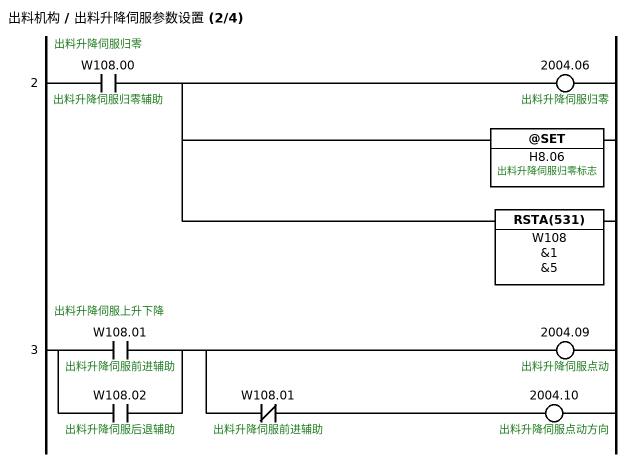
; [picture p360: 出料机构 / 出料升降伺服参数设置, rungs 2-3]
; rung 2: 出料升降伺服归零
LD W108.00  ; 出料升降伺服归零辅助
OUT 2004.06  ; 出料升降伺服归零
@SET H8.06  ; 出料升降伺服归零标志
RSTA(531) W108 &1 &5
; rung 3: 出料升降伺服上升下降
LD W108.01  ; 出料升降伺服前进辅助
OR W108.02  ; 出料升降伺服后退辅助
OUT 2004.09  ; 出料升降伺服点动
ANDNOT W108.01  ; 出料升降伺服前进辅助
OUT 2004.10  ; 出料升降伺服点动方向

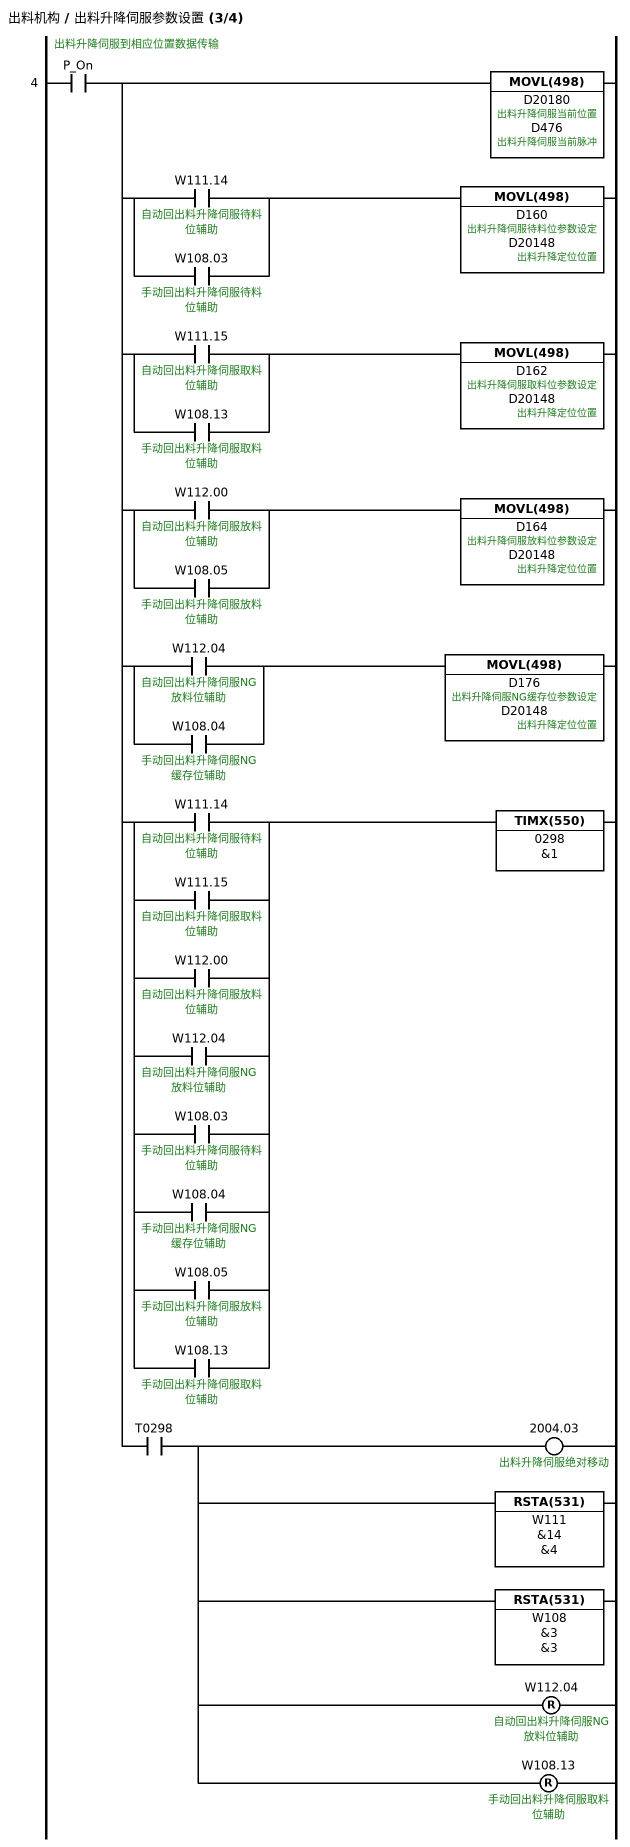
; rung 4: 出料升降伺服到相应位置数据传输
LD P_On
OUT TR0
MOVL(498) D20180 D476  ; 出料升降伺服当前位置, 出料升降伺服当前脉冲
LD W111.14  ; 自动回出料升降伺服待料位辅助
OR W108.03  ; 手动回出料升降伺服待料位辅助
ANDLD
MOVL(498) D160 D20148  ; 出料升降伺服待料位参数设定, 出料升降定位位置
LD TR0
LD W111.15  ; 自动回出料升降伺服取料位辅助
OR W108.13  ; 手动回出料升降伺服取料位辅助
ANDLD
MOVL(498) D162 D20148  ; 出料升降伺服取料位参数设定, 出料升降定位位置
LD TR0
LD W112.00  ; 自动回出料升降伺服放料位辅助
OR W108.05  ; 手动回出料升降伺服放料位辅助
ANDLD
MOVL(498) D164 D20148  ; 出料升降伺服放料位参数设定, 出料升降定位位置
LD TR0
LD W112.04  ; 自动回出料升降伺服NG放料位辅助
OR W108.04  ; 手动回出料升降伺服NG缓存位辅助
ANDLD
MOVL(498) D176 D20148  ; 出料升降伺服NG缓存位参数设定, 出料升降定位位置
LD TR0
LD W111.14  ; 自动回出料升降伺服待料位辅助
OR W111.15  ; 自动回出料升降伺服取料位辅助
OR W112.00  ; 自动回出料升降伺服放料位辅助
OR W112.04  ; 自动回出料升降伺服NG放料位辅助
OR W108.03  ; 手动回出料升降伺服待料位辅助
OR W108.04  ; 手动回出料升降伺服NG缓存位辅助
OR W108.05  ; 手动回出料升降伺服放料位辅助
OR W108.13  ; 手动回出料升降伺服取料位辅助
ANDLD
TIMX(550) 0298 &1
LD TR0
AND T0298
OUT 2004.03  ; 出料升降伺服绝对移动
RSTA(531) W111 &14 &4
RSTA(531) W108 &3 &3
RSET W112.04  ; 自动回出料升降伺服NG放料位辅助
RSET W108.13  ; 手动回出料升降伺服取料位辅助

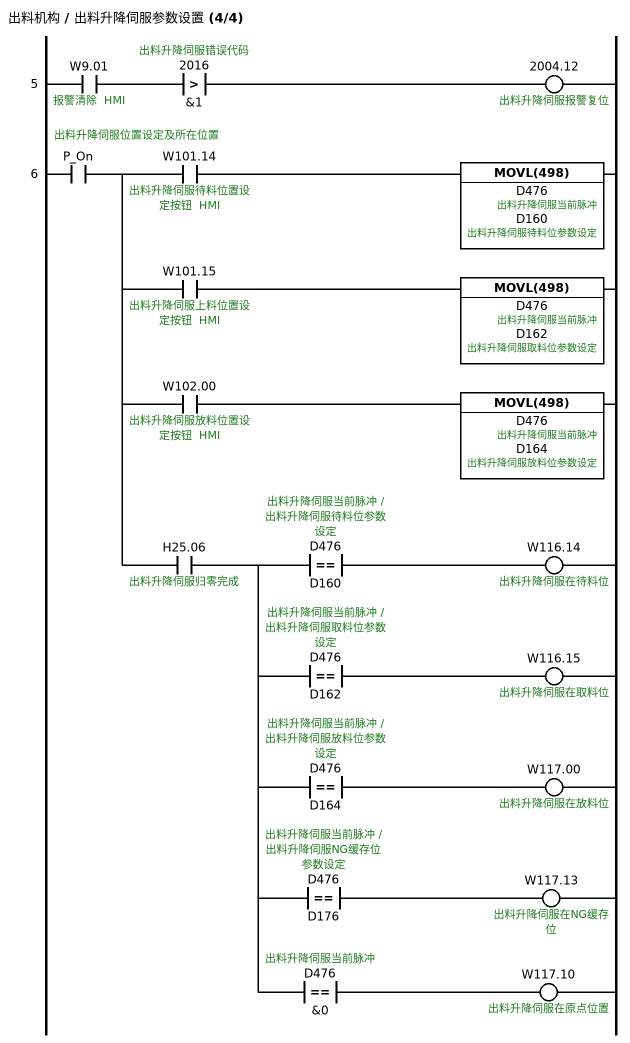
; rung 5
LD W9.01  ; 报警清除  HMI
AND>(320) 2016 &1  ; 出料升降伺服错误代码
OUT 2004.12  ; 出料升降伺服报警复位
; rung 6: 出料升降伺服位置设定及所在位置
LD P_On
OUT TR0
AND W101.14  ; 出料升降伺服待料位置设定按钮  HMI
MOVL(498) D476 D160  ; 出料升降伺服当前脉冲, 出料升降伺服待料位参数设定
LD TR0
AND W101.15  ; 出料升降伺服上料位置设定按钮  HMI
MOVL(498) D476 D162  ; 出料升降伺服当前脉冲, 出料升降伺服取料位参数设定
LD TR0
AND W102.00  ; 出料升降伺服放料位置设定按钮  HMI
MOVL(498) D476 D164  ; 出料升降伺服当前脉冲, 出料升降伺服放料位参数设定
LD TR0
AND H25.06  ; 出料升降伺服归零完成
OUT TR0
AND=SL(303) D476 D160  ; 出料升降伺服当前脉冲, 出料升降伺服待料位参数设定
OUT W116.14  ; 出料升降伺服在待料位
LD TR0
AND=SL(303) D476 D162  ; 出料升降伺服当前脉冲, 出料升降伺服取料位参数设定
OUT W116.15  ; 出料升降伺服在取料位
LD TR0
AND=SL(303) D476 D164  ; 出料升降伺服当前脉冲, 出料升降伺服放料位参数设定
OUT W117.00  ; 出料升降伺服在放料位
LD TR0
AND=SL(303) D476 D176  ; 出料升降伺服当前脉冲, 出料升降伺服NG缓存位参数设定
OUT W117.13  ; 出料升降伺服在NG缓存位
LD TR0
AND=SL(303) D476 &0  ; 出料升降伺服当前脉冲
OUT W117.10  ; 出料升降伺服在原点位置

### Section 出料旋转伺服参数设置

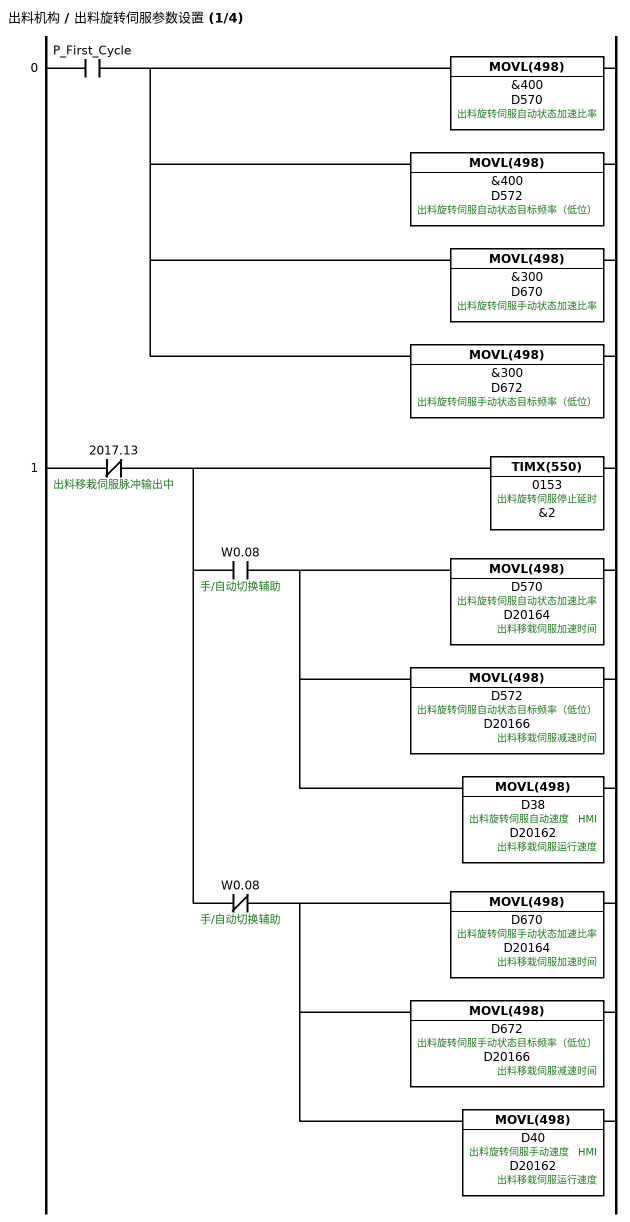
; rung 0
LD P_First_Cycle
MOVL(498) &400 D570  ; 出料旋转伺服自动状态加速比率
MOVL(498) &400 D572  ; 出料旋转伺服自动状态目标频率（低位）
MOVL(498) &300 D670  ; 出料旋转伺服手动状态加速比率
MOVL(498) &300 D672  ; 出料旋转伺服手动状态目标频率（低位）
; rung 1
LDNOT 2017.13  ; 出料移栽伺服脉冲输出中
OUT TR0
TIMX(550) 0153 &2  ; 出料旋转伺服停止延时
AND W0.08  ; 手/自动切换辅助
MOVL(498) D570 D20164  ; 出料旋转伺服自动状态加速比率, 出料移栽伺服加速时间
MOVL(498) D572 D20166  ; 出料旋转伺服自动状态目标频率（低位）, 出料移栽伺服减速时间
MOVL(498) D38 D20162  ; 出料旋转伺服自动速度   HMI, 出料移栽伺服运行速度
LD TR0
ANDNOT W0.08  ; 手/自动切换辅助
MOVL(498) D670 D20164  ; 出料旋转伺服手动状态加速比率, 出料移栽伺服加速时间
MOVL(498) D672 D20166  ; 出料旋转伺服手动状态目标频率（低位）, 出料移栽伺服减速时间
MOVL(498) D40 D20162  ; 出料旋转伺服手动速度   HMI, 出料移栽伺服运行速度

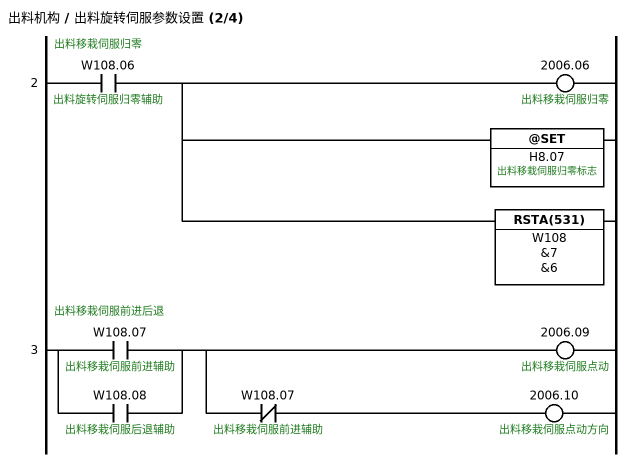
; rung 2: 出料移栽伺服归零
LD W108.06  ; 出料旋转伺服归零辅助
OUT 2006.06  ; 出料移栽伺服归零
@SET H8.07  ; 出料移栽伺服归零标志
RSTA(531) W108 &7 &6
; rung 3: 出料移栽伺服前进后退
LD W108.07  ; 出料移栽伺服前进辅助
OR W108.08  ; 出料移栽伺服后退辅助
OUT 2006.09  ; 出料移栽伺服点动
ANDNOT W108.07  ; 出料移栽伺服前进辅助
OUT 2006.10  ; 出料移栽伺服点动方向

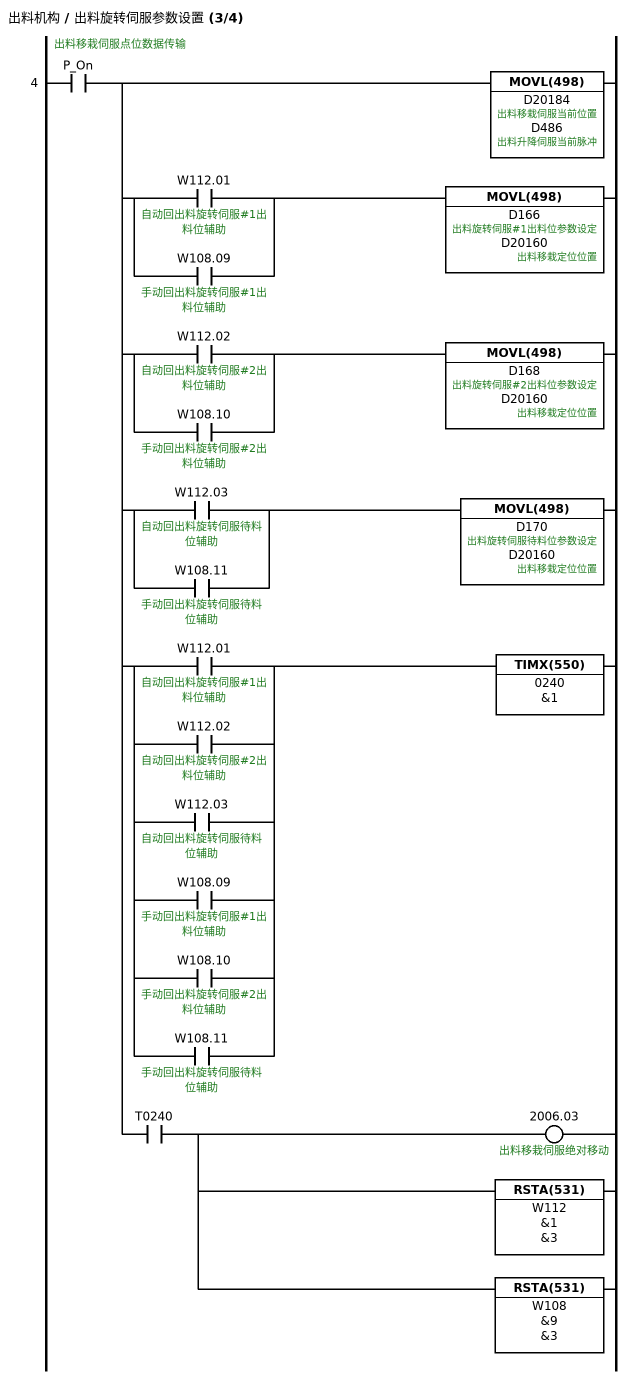
; rung 4: 出料移栽伺服点位数据传输
LD P_On
OUT TR0
MOVL(498) D20184 D486  ; 出料移栽伺服当前位置, 出料升降伺服当前脉冲
LD W112.01  ; 自动回出料旋转伺服#1出料位辅助
OR W108.09  ; 手动回出料旋转伺服#1出料位辅助
ANDLD
MOVL(498) D166 D20160  ; 出料旋转伺服#1出料位参数设定, 出料移栽定位位置
LD TR0
LD W112.02  ; 自动回出料旋转伺服#2出料位辅助
OR W108.10  ; 手动回出料旋转伺服#2出料位辅助
ANDLD
MOVL(498) D168 D20160  ; 出料旋转伺服#2出料位参数设定, 出料移栽定位位置
LD TR0
LD W112.03  ; 自动回出料旋转伺服待料位辅助
OR W108.11  ; 手动回出料旋转伺服待料位辅助
ANDLD
MOVL(498) D170 D20160  ; 出料旋转伺服待料位参数设定, 出料移栽定位位置
LD TR0
LD W112.01  ; 自动回出料旋转伺服#1出料位辅助
OR W112.02  ; 自动回出料旋转伺服#2出料位辅助
OR W112.03  ; 自动回出料旋转伺服待料位辅助
OR W108.09  ; 手动回出料旋转伺服#1出料位辅助
OR W108.10  ; 手动回出料旋转伺服#2出料位辅助
OR W108.11  ; 手动回出料旋转伺服待料位辅助
ANDLD
TIMX(550) 0240 &1
LD TR0
AND T0240
OUT 2006.03  ; 出料移栽伺服绝对移动
RSTA(531) W112 &1 &3
RSTA(531) W108 &9 &3

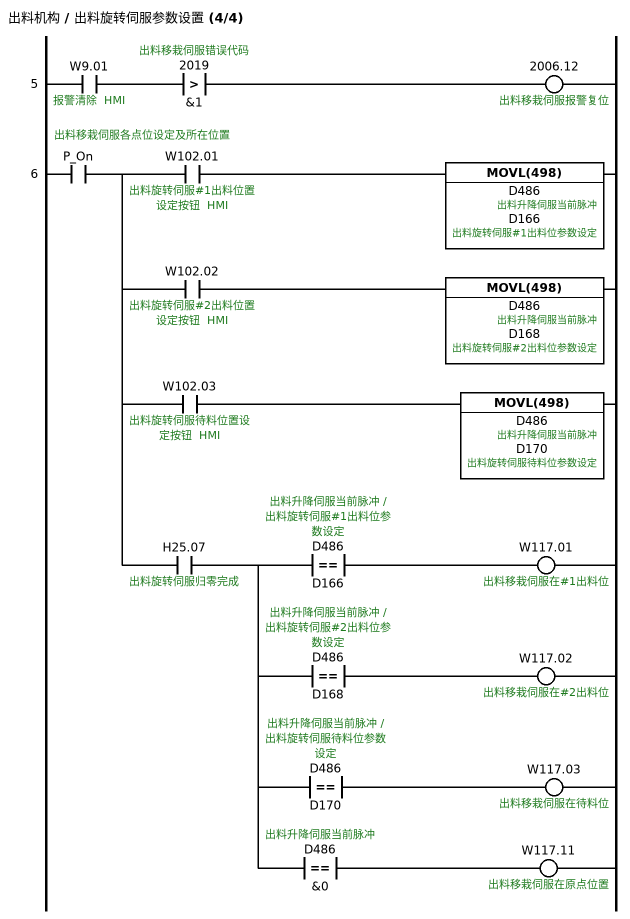
; rung 5
LD W9.01  ; 报警清除  HMI
AND>(320) 2019 &1  ; 出料移栽伺服错误代码
OUT 2006.12  ; 出料移栽伺服报警复位
; rung 6: 出料移栽伺服各点位设定及所在位置
LD P_On
OUT TR0
AND W102.01  ; 出料旋转伺服#1出料位置设定按钮  HMI
MOVL(498) D486 D166  ; 出料升降伺服当前脉冲, 出料旋转伺服#1出料位参数设定
LD TR0
AND W102.02  ; 出料旋转伺服#2出料位置设定按钮  HMI
MOVL(498) D486 D168  ; 出料升降伺服当前脉冲, 出料旋转伺服#2出料位参数设定
LD TR0
AND W102.03  ; 出料旋转伺服待料位置设定按钮  HMI
MOVL(498) D486 D170  ; 出料升降伺服当前脉冲, 出料旋转伺服待料位参数设定
LD TR0
AND H25.07  ; 出料旋转伺服归零完成
OUT TR0
AND=SL(303) D486 D166  ; 出料升降伺服当前脉冲, 出料旋转伺服#1出料位参数设定
OUT W117.01  ; 出料移栽伺服在#1出料位
LD TR0
AND=SL(303) D486 D168  ; 出料升降伺服当前脉冲, 出料旋转伺服#2出料位参数设定
OUT W117.02  ; 出料移栽伺服在#2出料位
LD TR0
AND=SL(303) D486 D170  ; 出料升降伺服当前脉冲, 出料旋转伺服待料位参数设定
OUT W117.03  ; 出料移栽伺服在待料位
LD TR0
AND=SL(303) D486 &0  ; 出料升降伺服当前脉冲
OUT W117.11  ; 出料移栽伺服在原点位置

### Section _4_框架信号对接

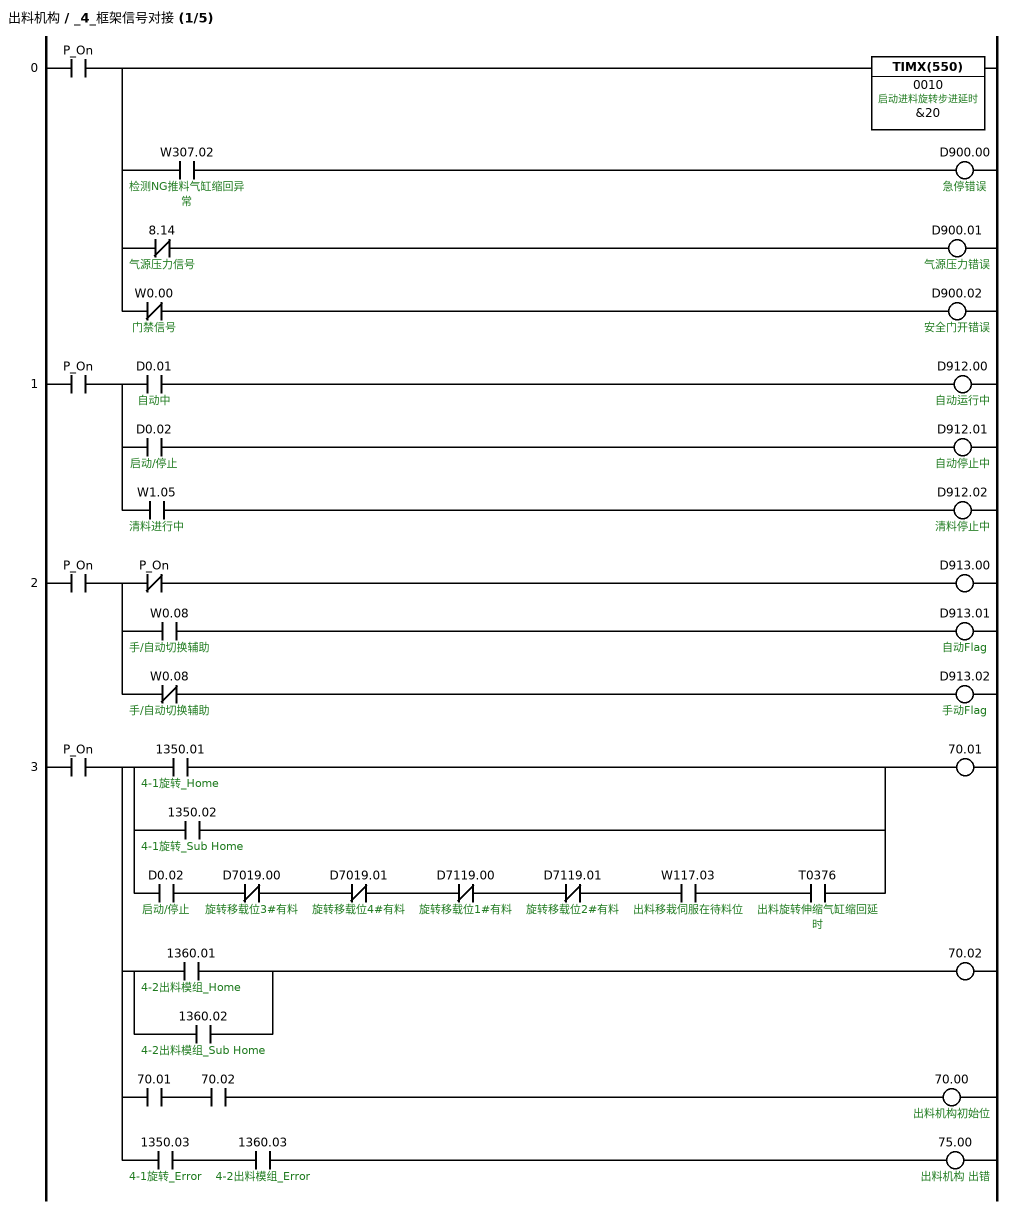
; rung 0
LD P_On
OUT TR0
TIMX(550) 0010 &20  ; 启动进料旋转步进延时
AND W307.02  ; 检测NG推料气缸缩回异常
OUT D900.00  ; 急停错误
LD TR0
ANDNOT 8.14  ; 气源压力信号
OUT D900.01  ; 气源压力错误
LD TR0
ANDNOT W0.00  ; 门禁信号
OUT D900.02  ; 安全门开错误
; rung 1
LD P_On
OUT TR0
AND D0.01  ; 自动中
OUT D912.00  ; 自动运行中
LD TR0
AND D0.02  ; 启动/停止
OUT D912.01  ; 自动停止中
LD TR0
AND W1.05  ; 清料进行中
OUT D912.02  ; 清料停止中
; rung 2
LD P_On
OUT TR0
ANDNOT P_On
OUT D913.00
LD TR0
AND W0.08  ; 手/自动切换辅助
OUT D913.01  ; 自动Flag
LD TR0
ANDNOT W0.08  ; 手/自动切换辅助
OUT D913.02  ; 手动Flag
; rung 3
LD P_On
OUT TR0
LD 1350.01  ; 4-1旋转_Home
OR 1350.02  ; 4-1旋转_Sub Home
LD D0.02  ; 启动/停止
ANDNOT D7019.00  ; 旋转移载位3#有料
ANDNOT D7019.01  ; 旋转移载位4#有料
ANDNOT D7119.00  ; 旋转移载位1#有料
ANDNOT D7119.01  ; 旋转移载位2#有料
AND W117.03  ; 出料移栽伺服在待料位
AND T0376  ; 出料旋转伸缩气缸缩回延时
ORLD
ANDLD
OUT 70.01
LD TR0
LD 1360.01  ; 4-2出料模组_Home
OR 1360.02  ; 4-2出料模组_Sub Home
ANDLD
OUT 70.02
LD TR0
AND 70.01
AND 70.02
OUT 70.00  ; 出料机构初始位
LD TR0
AND 1350.03  ; 4-1旋转_Error
AND 1360.03  ; 4-2出料模组_Error
OUT 75.00  ; 出料机构 出错

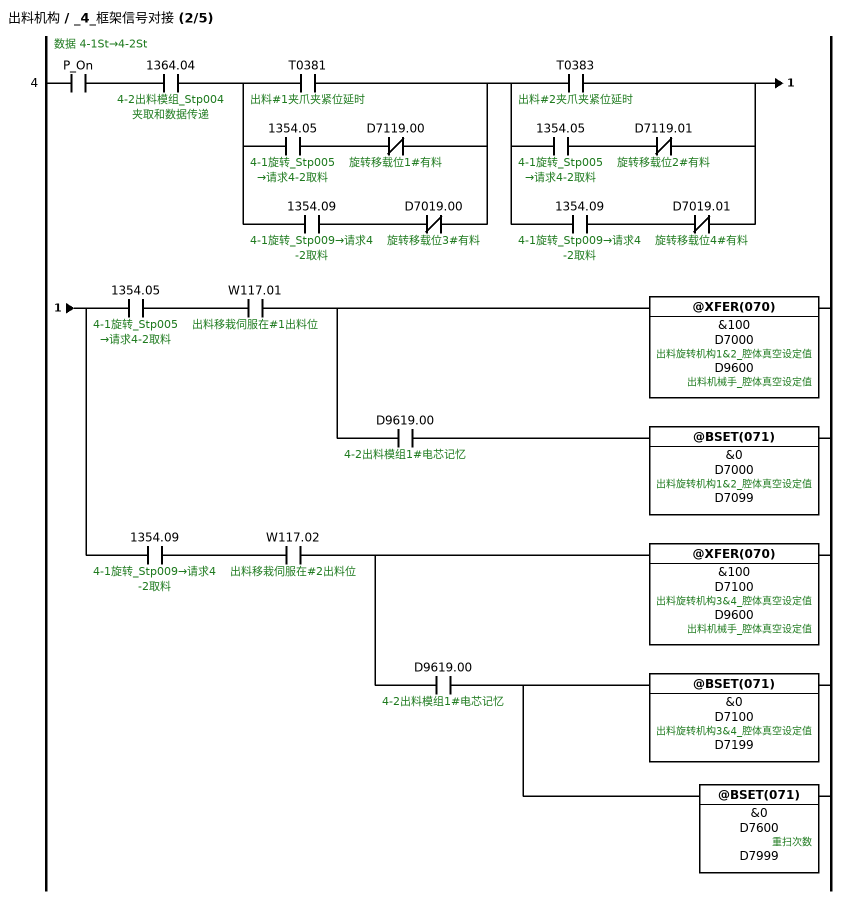
; rung 4: 数据 4-1St→4-2St
LD P_On
AND 1364.04  ; 4-2出料模组_Stp004 夹取和数据传递
LD T0381  ; 出料#1夹爪夹紧位延时
LD 1354.05  ; 4-1旋转_Stp005 →请求4-2取料
ANDNOT D7119.00  ; 旋转移载位1#有料
ORLD
LD 1354.09  ; 4-1旋转_Stp009→请求4-2取料
ANDNOT D7019.00  ; 旋转移载位3#有料
ORLD
ANDLD
LD T0383  ; 出料#2夹爪夹紧位延时
LD 1354.05  ; 4-1旋转_Stp005 →请求4-2取料
ANDNOT D7119.01  ; 旋转移载位2#有料
ORLD
LD 1354.09  ; 4-1旋转_Stp009→请求4-2取料
ANDNOT D7019.01  ; 旋转移载位4#有料
ORLD
ANDLD
OUT TR0
AND 1354.05  ; 4-1旋转_Stp005 →请求4-2取料
AND W117.01  ; 出料移栽伺服在#1出料位
@XFER(070) &100 D7000 D9600  ; 出料旋转机构1&2_腔体真空设定值, 出料机械手_腔体真空设定值
AND D9619.00  ; 4-2出料模组1#电芯记忆
@BSET(071) &0 D7000 D7099  ; 出料旋转机构1&2_腔体真空设定值
LD TR0
AND 1354.09  ; 4-1旋转_Stp009→请求4-2取料
AND W117.02  ; 出料移栽伺服在#2出料位
@XFER(070) &100 D7100 D9600  ; 出料旋转机构3&4_腔体真空设定值, 出料机械手_腔体真空设定值
AND D9619.00  ; 4-2出料模组1#电芯记忆
@BSET(071) &0 D7100 D7199  ; 出料旋转机构3&4_腔体真空设定值
@BSET(071) &0 D7600 D7999  ; 重扫次数

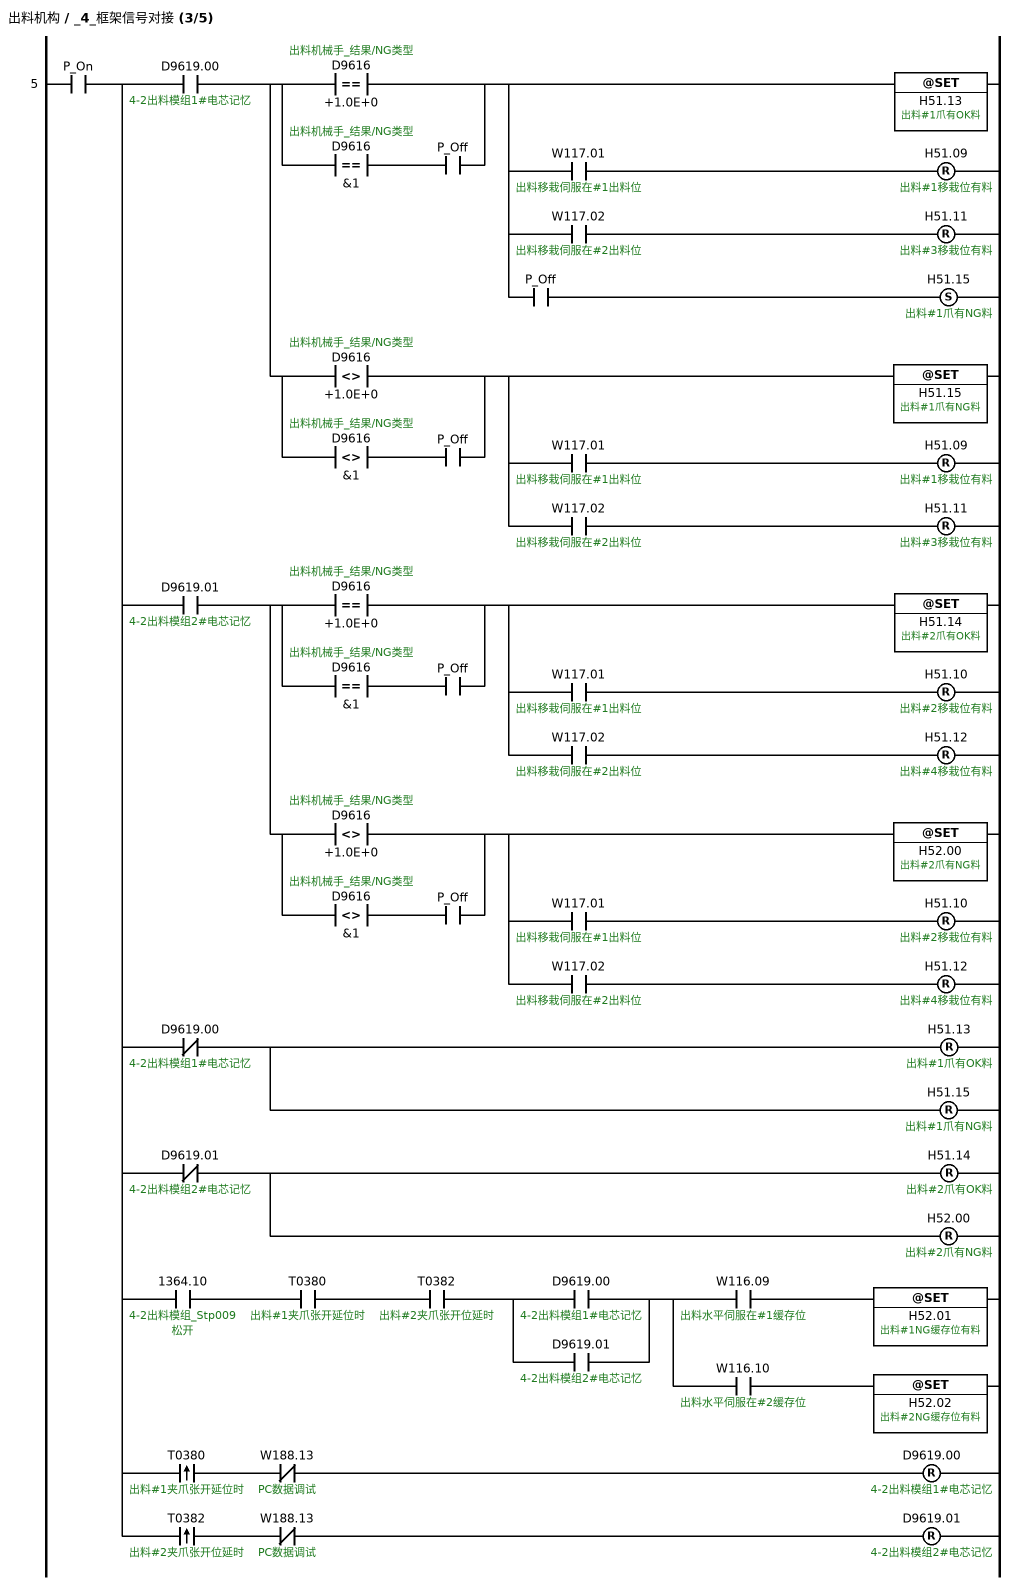
; rung 5
LD P_On
OUT TR0
AND D9619.00  ; 4-2出料模组1#电芯记忆
OUT TR1
LD=F(329) D9616 +1.0E+0  ; 出料机械手_结果/NG类型
LD=(300) D9616 &1  ; 出料机械手_结果/NG类型
AND P_Off
ORLD
ANDLD
OUT TR2
@SET H51.13  ; 出料#1爪有OK料
AND W117.01  ; 出料移栽伺服在#1出料位
RSET H51.09  ; 出料#1移栽位有料
LD TR2
AND W117.02  ; 出料移栽伺服在#2出料位
RSET H51.11  ; 出料#3移栽位有料
LD TR2
AND P_Off
SET H51.15  ; 出料#1爪有NG料
LD TR1
LD<>F(330) D9616 +1.0E+0  ; 出料机械手_结果/NG类型
LD<>(305) D9616 &1  ; 出料机械手_结果/NG类型
AND P_Off
ORLD
ANDLD
OUT TR1
@SET H51.15  ; 出料#1爪有NG料
AND W117.01  ; 出料移栽伺服在#1出料位
RSET H51.09  ; 出料#1移栽位有料
LD TR1
AND W117.02  ; 出料移栽伺服在#2出料位
RSET H51.11  ; 出料#3移栽位有料
LD TR0
AND D9619.01  ; 4-2出料模组2#电芯记忆
OUT TR1
LD=F(329) D9616 +1.0E+0  ; 出料机械手_结果/NG类型
LD=(300) D9616 &1  ; 出料机械手_结果/NG类型
AND P_Off
ORLD
ANDLD
OUT TR2
@SET H51.14  ; 出料#2爪有OK料
AND W117.01  ; 出料移栽伺服在#1出料位
RSET H51.10  ; 出料#2移栽位有料
LD TR2
AND W117.02  ; 出料移栽伺服在#2出料位
RSET H51.12  ; 出料#4移栽位有料
LD TR1
LD<>F(330) D9616 +1.0E+0  ; 出料机械手_结果/NG类型
LD<>(305) D9616 &1  ; 出料机械手_结果/NG类型
AND P_Off
ORLD
ANDLD
OUT TR1
@SET H52.00  ; 出料#2爪有NG料
AND W117.01  ; 出料移栽伺服在#1出料位
RSET H51.10  ; 出料#2移栽位有料
LD TR1
AND W117.02  ; 出料移栽伺服在#2出料位
RSET H51.12  ; 出料#4移栽位有料
LD TR0
ANDNOT D9619.00  ; 4-2出料模组1#电芯记忆
RSET H51.13  ; 出料#1爪有OK料
RSET H51.15  ; 出料#1爪有NG料
LD TR0
ANDNOT D9619.01  ; 4-2出料模组2#电芯记忆
RSET H51.14  ; 出料#2爪有OK料
RSET H52.00  ; 出料#2爪有NG料
LD TR0
AND 1364.10  ; 4-2出料模组_Stp009 松开
AND T0380  ; 出料#1夹爪张开延位时
AND T0382  ; 出料#2夹爪张开位延时
LD D9619.00  ; 4-2出料模组1#电芯记忆
OR D9619.01  ; 4-2出料模组2#电芯记忆
ANDLD
OUT TR1
AND W116.09  ; 出料水平伺服在#1缓存位
@SET H52.01  ; 出料#1NG缓存位有料
LD TR1
AND W116.10  ; 出料水平伺服在#2缓存位
@SET H52.02  ; 出料#2NG缓存位有料
LD TR0
@AND T0380  ; 出料#1夹爪张开延位时
ANDNOT W188.13  ; PC数据调试
RSET D9619.00  ; 4-2出料模组1#电芯记忆
LD TR0
@AND T0382  ; 出料#2夹爪张开位延时
ANDNOT W188.13  ; PC数据调试
RSET D9619.01  ; 4-2出料模组2#电芯记忆

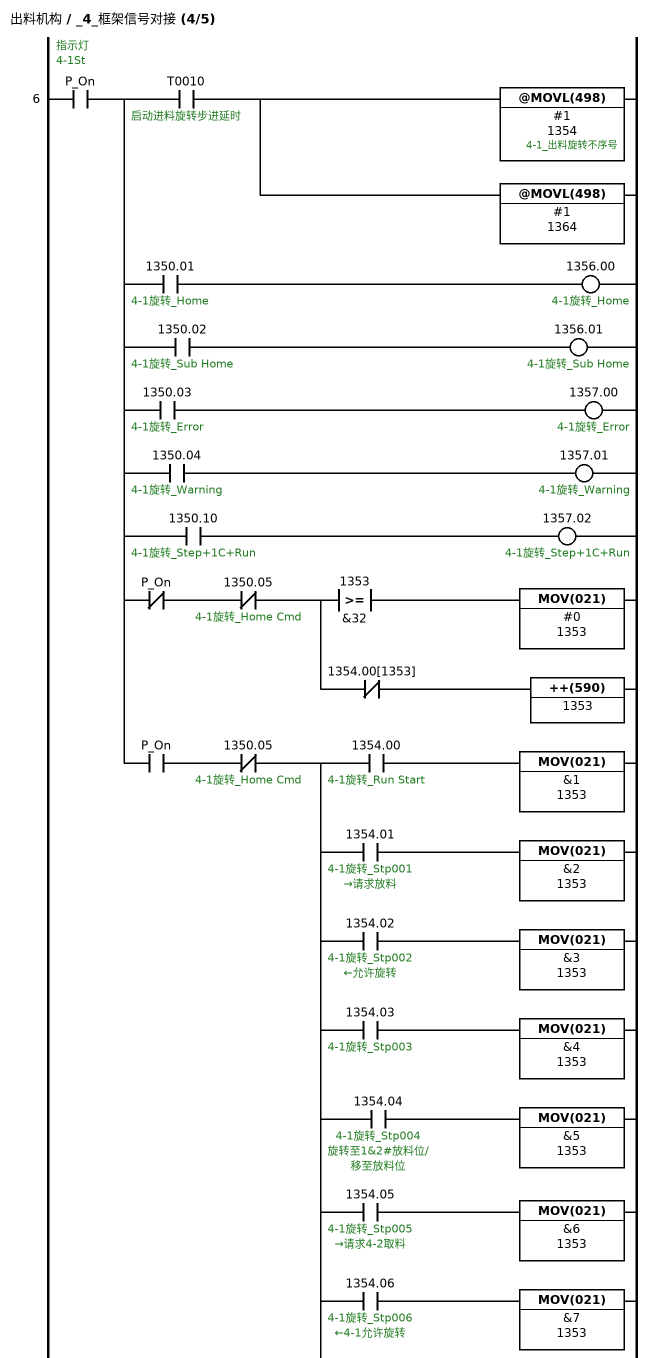

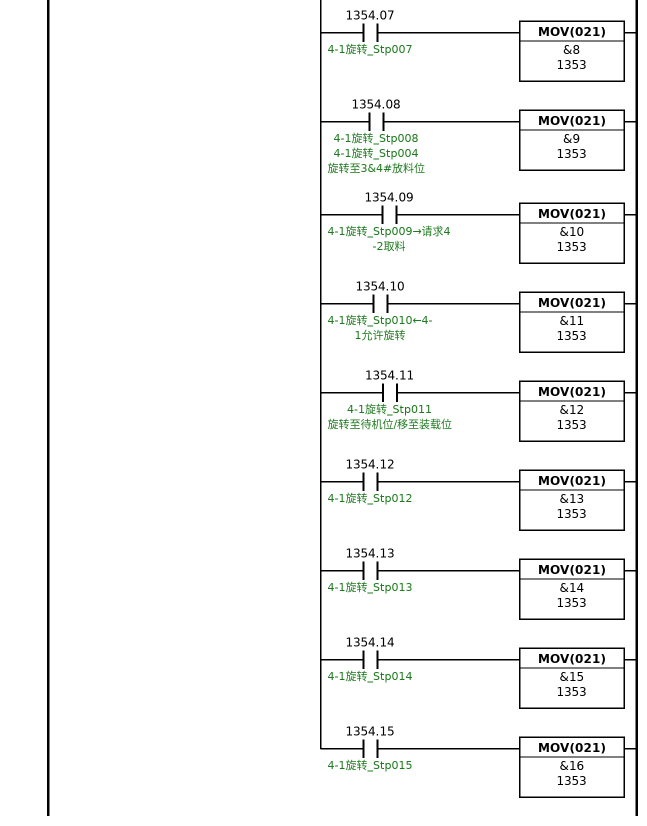
; rung 6: 指示灯 / 4-1St
LD P_On
OUT TR0
AND T0010  ; 启动进料旋转步进延时
@MOVL(498) #1 1354  ; 4-1_出料旋转不序号
@MOVL(498) #1 1364
LD TR0
AND 1350.01  ; 4-1旋转_Home
OUT 1356.00  ; 4-1旋转_Home
LD TR0
AND 1350.02  ; 4-1旋转_Sub Home
OUT 1356.01  ; 4-1旋转_Sub Home
LD TR0
AND 1350.03  ; 4-1旋转_Error
OUT 1357.00  ; 4-1旋转_Error
LD TR0
AND 1350.04  ; 4-1旋转_Warning
OUT 1357.01  ; 4-1旋转_Warning
LD TR0
AND 1350.10  ; 4-1旋转_Step+1C+Run
OUT 1357.02  ; 4-1旋转_Step+1C+Run
LD TR0
ANDNOT P_On
ANDNOT 1350.05  ; 4-1旋转_Home Cmd
OUT TR1
AND>=(325) 1353 &32
MOV(021) #0 1353
LD TR1
ANDNOT 1354.00[1353]
++(590) 1353
LD TR0
AND P_On
ANDNOT 1350.05  ; 4-1旋转_Home Cmd
OUT TR0
AND 1354.00  ; 4-1旋转_Run Start
MOV(021) &1 1353
LD TR0
AND 1354.01  ; 4-1旋转_Stp001 →请求放料
MOV(021) &2 1353
LD TR0
AND 1354.02  ; 4-1旋转_Stp002 ←允许旋转
MOV(021) &3 1353
LD TR0
AND 1354.03  ; 4-1旋转_Stp003
MOV(021) &4 1353
LD TR0
AND 1354.04  ; 4-1旋转_Stp004 旋转至1&2#放料位/移至放料位
MOV(021) &5 1353
LD TR0
AND 1354.05  ; 4-1旋转_Stp005 →请求4-2取料
MOV(021) &6 1353
LD TR0
AND 1354.06  ; 4-1旋转_Stp006 ←4-1允许旋转
MOV(021) &7 1353
LD TR0
AND 1354.07  ; 4-1旋转_Stp007
MOV(021) &8 1353
LD TR0
AND 1354.08  ; 4-1旋转_Stp008 4-1旋转_Stp004 旋转至3&4#放料位
MOV(021) &9 1353
LD TR0
AND 1354.09  ; 4-1旋转_Stp009→请求4-2取料
MOV(021) &10 1353
LD TR0
AND 1354.10  ; 4-1旋转_Stp010←4-1允许旋转
MOV(021) &11 1353
LD TR0
AND 1354.11  ; 4-1旋转_Stp011 旋转至待机位/移至装载位
MOV(021) &12 1353
LD TR0
AND 1354.12  ; 4-1旋转_Stp012
MOV(021) &13 1353
LD TR0
AND 1354.13  ; 4-1旋转_Stp013
MOV(021) &14 1353
LD TR0
AND 1354.14  ; 4-1旋转_Stp014
MOV(021) &15 1353
LD TR0
AND 1354.15  ; 4-1旋转_Stp015
MOV(021) &16 1353

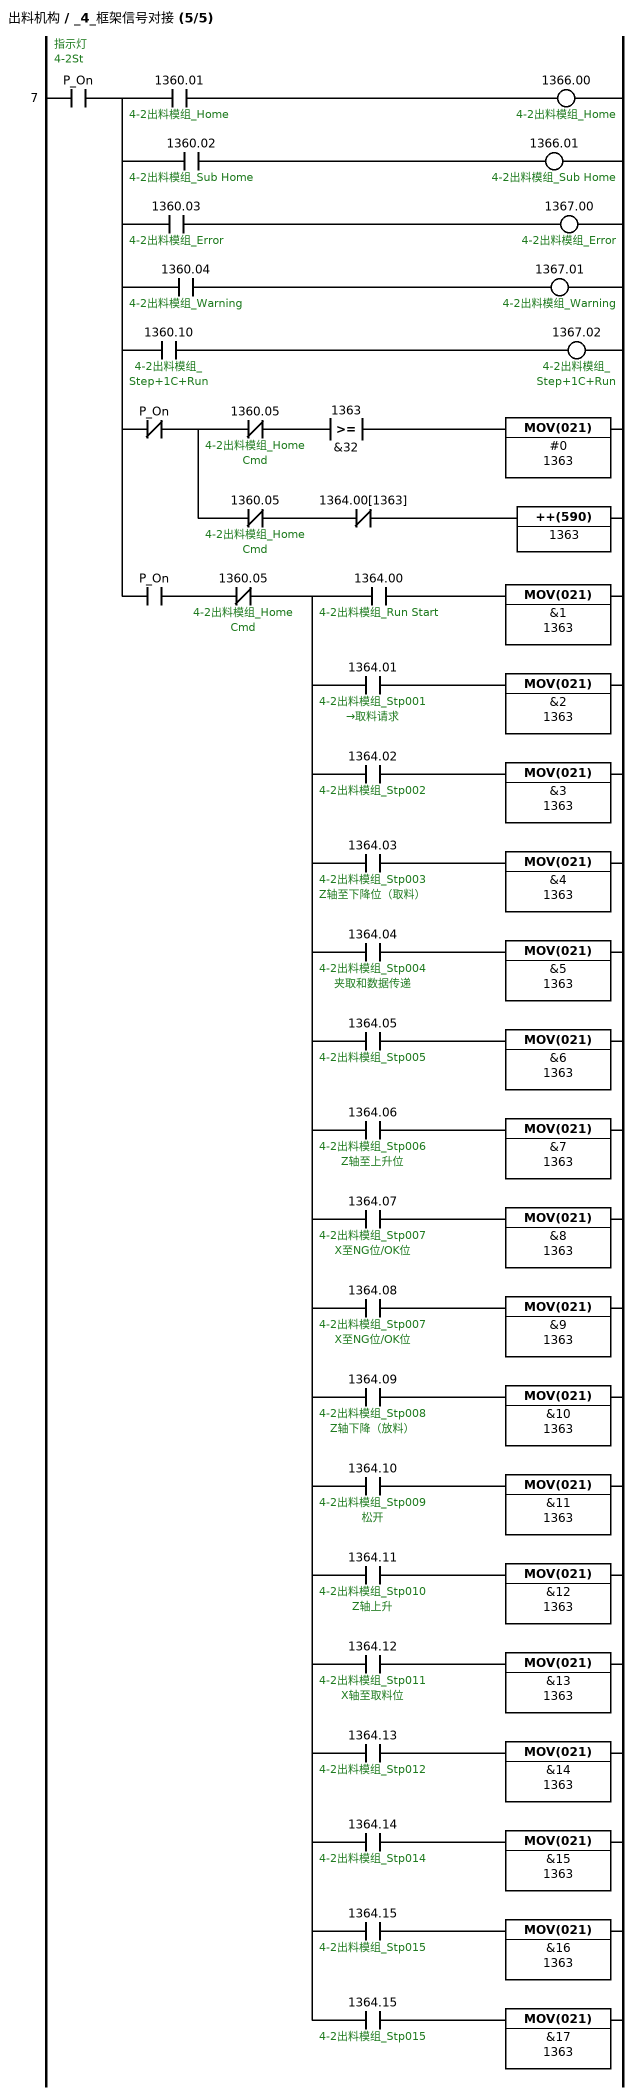
; rung 7: 指示灯 / 4-2St
LD P_On
OUT TR0
AND 1360.01  ; 4-2出料模组_Home
OUT 1366.00  ; 4-2出料模组_Home
LD TR0
AND 1360.02  ; 4-2出料模组_Sub Home
OUT 1366.01  ; 4-2出料模组_Sub Home
LD TR0
AND 1360.03  ; 4-2出料模组_Error
OUT 1367.00  ; 4-2出料模组_Error
LD TR0
AND 1360.04  ; 4-2出料模组_Warning
OUT 1367.01  ; 4-2出料模组_Warning
LD TR0
AND 1360.10  ; 4-2出料模组_Step+1C+Run
OUT 1367.02  ; 4-2出料模组_Step+1C+Run
LD TR0
ANDNOT P_On
OUT TR1
ANDNOT 1360.05  ; 4-2出料模组_Home Cmd
AND>=(325) 1363 &32
MOV(021) #0 1363
LD TR1
ANDNOT 1360.05  ; 4-2出料模组_Home Cmd
ANDNOT 1364.00[1363]
++(590) 1363
LD TR0
AND P_On
ANDNOT 1360.05  ; 4-2出料模组_Home Cmd
OUT TR0
AND 1364.00  ; 4-2出料模组_Run Start
MOV(021) &1 1363
LD TR0
AND 1364.01  ; 4-2出料模组_Stp001 →取料请求
MOV(021) &2 1363
LD TR0
AND 1364.02  ; 4-2出料模组_Stp002
MOV(021) &3 1363
LD TR0
AND 1364.03  ; 4-2出料模组_Stp003 Z轴至下降位（取料）
MOV(021) &4 1363
LD TR0
AND 1364.04  ; 4-2出料模组_Stp004 夹取和数据传递
MOV(021) &5 1363
LD TR0
AND 1364.05  ; 4-2出料模组_Stp005
MOV(021) &6 1363
LD TR0
AND 1364.06  ; 4-2出料模组_Stp006 Z轴至上升位
MOV(021) &7 1363
LD TR0
AND 1364.07  ; 4-2出料模组_Stp007 X至NG位/OK位
MOV(021) &8 1363
LD TR0
AND 1364.08  ; 4-2出料模组_Stp007 X至NG位/OK位
MOV(021) &9 1363
LD TR0
AND 1364.09  ; 4-2出料模组_Stp008 Z轴下降（放料）
MOV(021) &10 1363
LD TR0
AND 1364.10  ; 4-2出料模组_Stp009 松开
MOV(021) &11 1363
LD TR0
AND 1364.11  ; 4-2出料模组_Stp010 Z轴上升
MOV(021) &12 1363
LD TR0
AND 1364.12  ; 4-2出料模组_Stp011 X轴至取料位
MOV(021) &13 1363
LD TR0
AND 1364.13  ; 4-2出料模组_Stp012
MOV(021) &14 1363
LD TR0
AND 1364.14  ; 4-2出料模组_Stp014
MOV(021) &15 1363
LD TR0
AND 1364.15  ; 4-2出料模组_Stp015
MOV(021) &16 1363
LD TR0
AND 1364.15  ; 4-2出料模组_Stp015
MOV(021) &17 1363

### Section _4_1出料旋转自动

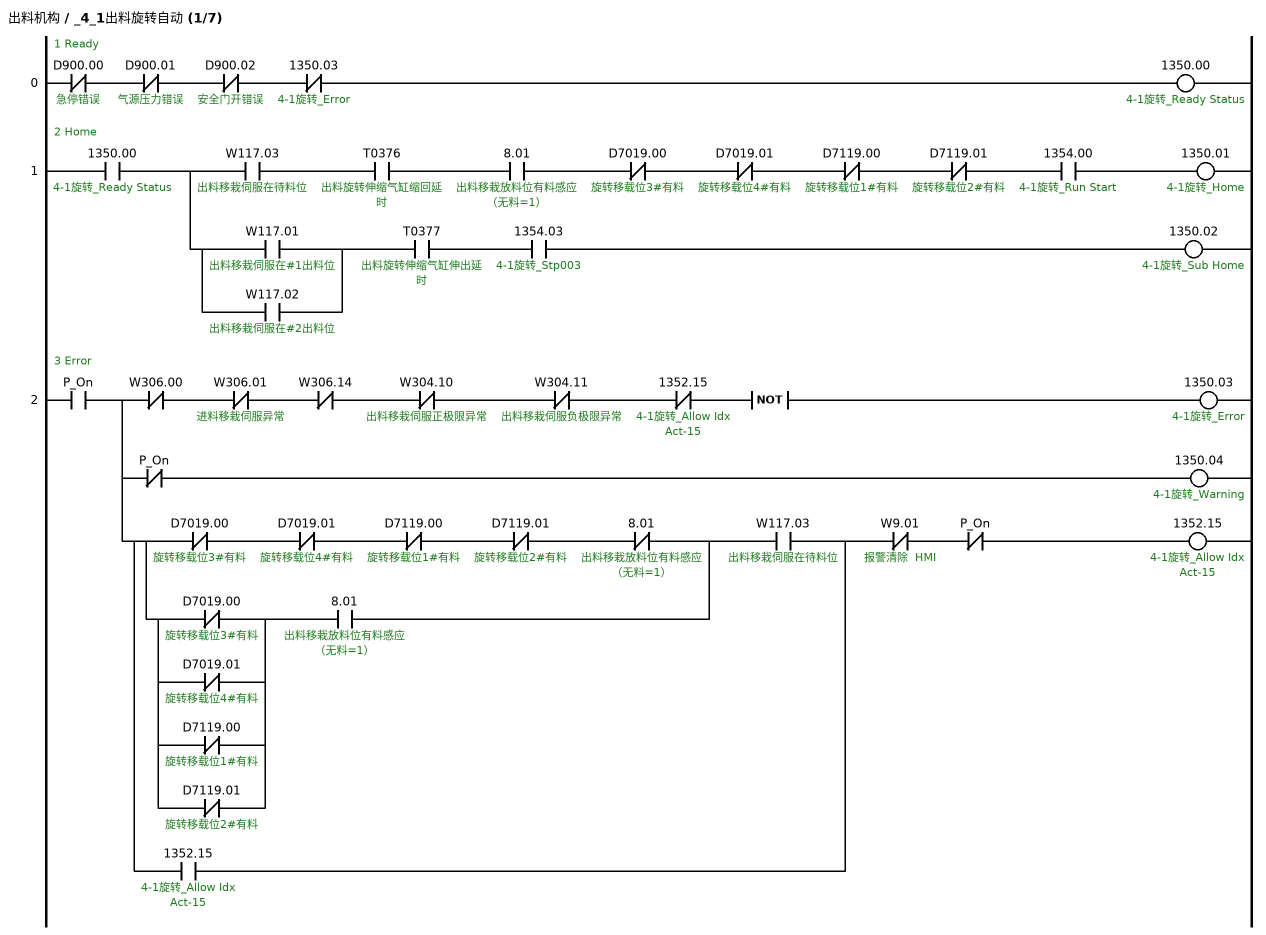
; rung 0: 1 Ready
LDNOT D900.00  ; 急停错误
ANDNOT D900.01  ; 气源压力错误
ANDNOT D900.02  ; 安全门开错误
ANDNOT 1350.03  ; 4-1旋转_Error
OUT 1350.00  ; 4-1旋转_Ready Status
; rung 1: 2 Home
LD 1350.00  ; 4-1旋转_Ready Status
OUT TR0
AND W117.03  ; 出料移栽伺服在待料位
AND T0376  ; 出料旋转伸缩气缸缩回延时
AND 8.01  ; 出料移栽放料位有料感应（无料=1）
ANDNOT D7019.00  ; 旋转移载位3#有料
ANDNOT D7019.01  ; 旋转移载位4#有料
ANDNOT D7119.00  ; 旋转移载位1#有料
ANDNOT D7119.01  ; 旋转移载位2#有料
AND 1354.00  ; 4-1旋转_Run Start
OUT 1350.01  ; 4-1旋转_Home
LD TR0
LD W117.01  ; 出料移栽伺服在#1出料位
OR W117.02  ; 出料移栽伺服在#2出料位
ANDLD
AND T0377  ; 出料旋转伸缩气缸伸出延时
AND 1354.03  ; 4-1旋转_Stp003
OUT 1350.02  ; 4-1旋转_Sub Home
; rung 2: 3 Error
LD P_On
OUT TR0
ANDNOT W306.00
ANDNOT W306.01  ; 进料移栽伺服异常
ANDNOT W306.14
ANDNOT W304.10  ; 出料移栽伺服正极限异常
ANDNOT W304.11  ; 出料移栽伺服负极限异常
ANDNOT 1352.15  ; 4-1旋转_Allow Idx Act-15
NOT(520)
OUT 1350.03  ; 4-1旋转_Error
LD TR0
ANDNOT P_On
OUT 1350.04  ; 4-1旋转_Warning
LD TR0
LDNOT D7019.00  ; 旋转移载位3#有料
ANDNOT D7019.01  ; 旋转移载位4#有料
ANDNOT D7119.00  ; 旋转移载位1#有料
ANDNOT D7119.01  ; 旋转移载位2#有料
ANDNOT 8.01  ; 出料移栽放料位有料感应（无料=1）
LDNOT D7019.00  ; 旋转移载位3#有料
ORNOT D7019.01  ; 旋转移载位4#有料
ORNOT D7119.00  ; 旋转移载位1#有料
ORNOT D7119.01  ; 旋转移载位2#有料
AND 8.01  ; 出料移栽放料位有料感应（无料=1）
ORLD
AND W117.03  ; 出料移栽伺服在待料位
OR 1352.15  ; 4-1旋转_Allow Idx Act-15
ANDLD
ANDNOT W9.01  ; 报警清除  HMI
ANDNOT P_On
OUT 1352.15  ; 4-1旋转_Allow Idx Act-15

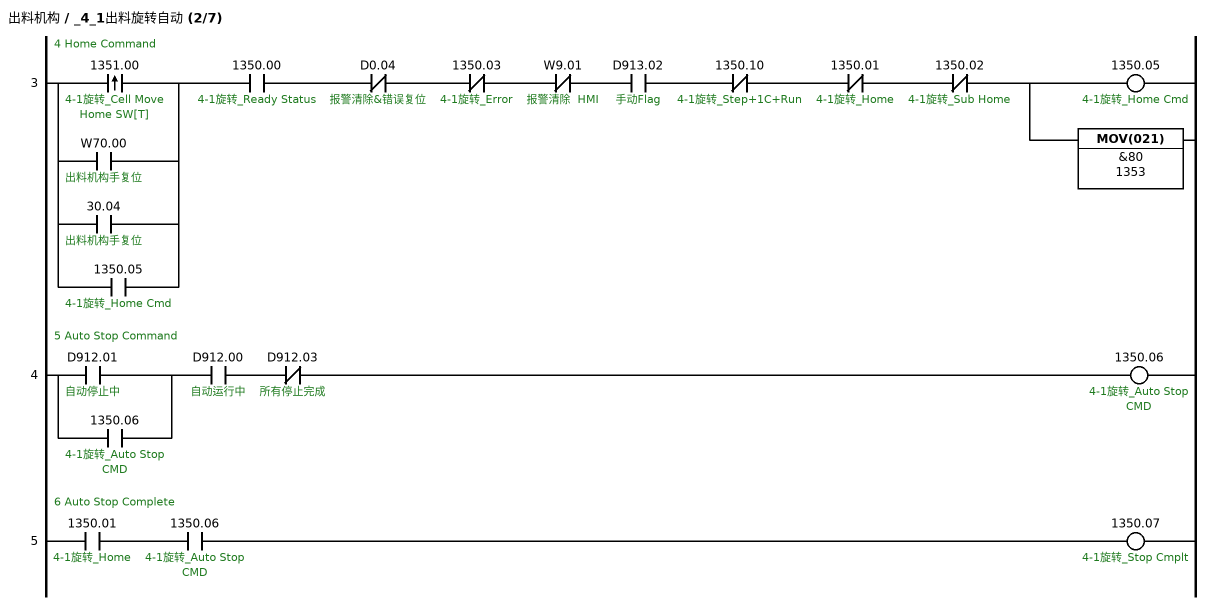
; rung 3: 4 Home Command
@LD 1351.00  ; 4-1旋转_Cell Move Home SW[T]
OR W70.00  ; 出料机构手复位
OR 30.04  ; 出料机构手复位
OR 1350.05  ; 4-1旋转_Home Cmd
AND 1350.00  ; 4-1旋转_Ready Status
ANDNOT D0.04  ; 报警清除&错误复位
ANDNOT 1350.03  ; 4-1旋转_Error
ANDNOT W9.01  ; 报警清除  HMI
AND D913.02  ; 手动Flag
ANDNOT 1350.10  ; 4-1旋转_Step+1C+Run
ANDNOT 1350.01  ; 4-1旋转_Home
ANDNOT 1350.02  ; 4-1旋转_Sub Home
OUT 1350.05  ; 4-1旋转_Home Cmd
MOV(021) &80 1353
; rung 4: 5 Auto Stop Command
LD D912.01  ; 自动停止中
OR 1350.06  ; 4-1旋转_Auto Stop CMD
AND D912.00  ; 自动运行中
ANDNOT D912.03  ; 所有停止完成
OUT 1350.06  ; 4-1旋转_Auto Stop CMD
; rung 5: 6 Auto Stop Complete
LD 1350.01  ; 4-1旋转_Home
AND 1350.06  ; 4-1旋转_Auto Stop CMD
OUT 1350.07  ; 4-1旋转_Stop Cmplt

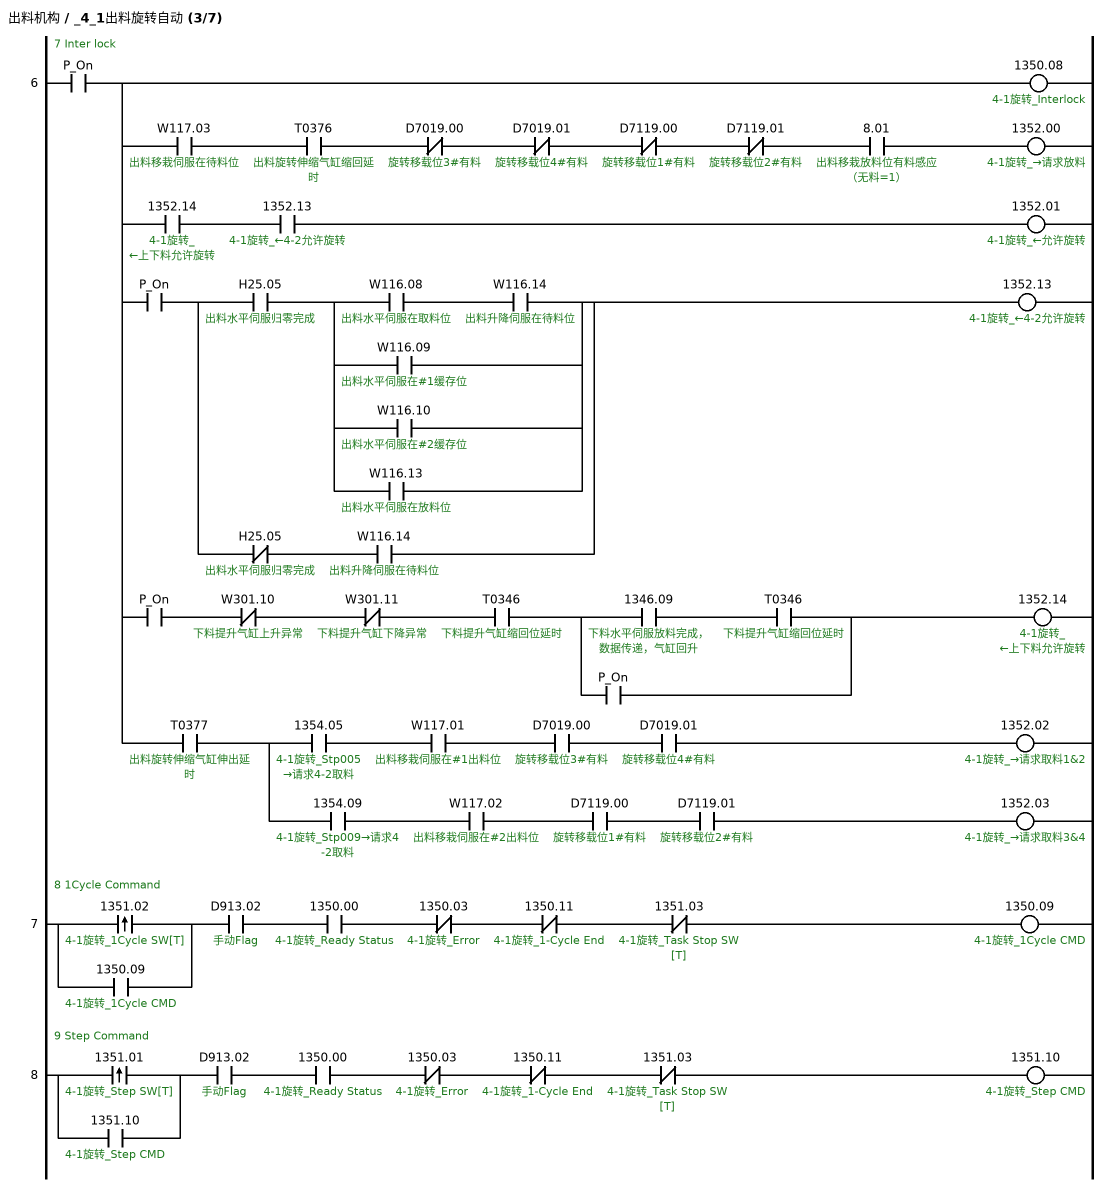
; rung 6: 7 Inter lock
LD P_On
OUT TR0
OUT 1350.08  ; 4-1旋转_Interlock
AND W117.03  ; 出料移栽伺服在待料位
AND T0376  ; 出料旋转伸缩气缸缩回延时
ANDNOT D7019.00  ; 旋转移载位3#有料
ANDNOT D7019.01  ; 旋转移载位4#有料
ANDNOT D7119.00  ; 旋转移载位1#有料
ANDNOT D7119.01  ; 旋转移载位2#有料
AND 8.01  ; 出料移栽放料位有料感应（无料=1）
OUT 1352.00  ; 4-1旋转_→请求放料
LD TR0
AND 1352.14  ; 4-1旋转_←上下料允许旋转
AND 1352.13  ; 4-1旋转_←4-2允许旋转
OUT 1352.01  ; 4-1旋转_←允许旋转
LD TR0
AND P_On
LD H25.05  ; 出料水平伺服归零完成
LD W116.08  ; 出料水平伺服在取料位
AND W116.14  ; 出料升降伺服在待料位
OR W116.09  ; 出料水平伺服在#1缓存位
OR W116.10  ; 出料水平伺服在#2缓存位
OR W116.13  ; 出料水平伺服在放料位
ANDLD
LDNOT H25.05  ; 出料水平伺服归零完成
AND W116.14  ; 出料升降伺服在待料位
ORLD
ANDLD
OUT 1352.13  ; 4-1旋转_←4-2允许旋转
LD TR0
AND P_On
ANDNOT W301.10  ; 下料提升气缸上升异常
ANDNOT W301.11  ; 下料提升气缸下降异常
AND T0346  ; 下料提升气缸缩回位延时
LD 1346.09  ; 下料水平伺服放料完成，数据传递，气缸回升
AND T0346  ; 下料提升气缸缩回位延时
OR P_On
ANDLD
OUT 1352.14  ; 4-1旋转_←上下料允许旋转
LD TR0
AND T0377  ; 出料旋转伸缩气缸伸出延时
OUT TR0
AND 1354.05  ; 4-1旋转_Stp005 →请求4-2取料
AND W117.01  ; 出料移栽伺服在#1出料位
AND D7019.00  ; 旋转移载位3#有料
AND D7019.01  ; 旋转移载位4#有料
OUT 1352.02  ; 4-1旋转_→请求取料1&2
LD TR0
AND 1354.09  ; 4-1旋转_Stp009→请求4-2取料
AND W117.02  ; 出料移栽伺服在#2出料位
AND D7119.00  ; 旋转移载位1#有料
AND D7119.01  ; 旋转移载位2#有料
OUT 1352.03  ; 4-1旋转_→请求取料3&4
; rung 7: 8 1Cycle Command
@LD 1351.02  ; 4-1旋转_1Cycle SW[T]
OR 1350.09  ; 4-1旋转_1Cycle CMD
AND D913.02  ; 手动Flag
AND 1350.00  ; 4-1旋转_Ready Status
ANDNOT 1350.03  ; 4-1旋转_Error
ANDNOT 1350.11  ; 4-1旋转_1-Cycle End
ANDNOT 1351.03  ; 4-1旋转_Task Stop SW [T]
OUT 1350.09  ; 4-1旋转_1Cycle CMD
; rung 8: 9 Step Command
@LD 1351.01  ; 4-1旋转_Step SW[T]
OR 1351.10  ; 4-1旋转_Step CMD
AND D913.02  ; 手动Flag
AND 1350.00  ; 4-1旋转_Ready Status
ANDNOT 1350.03  ; 4-1旋转_Error
ANDNOT 1350.11  ; 4-1旋转_1-Cycle End
ANDNOT 1351.03  ; 4-1旋转_Task Stop SW [T]
OUT 1351.10  ; 4-1旋转_Step CMD

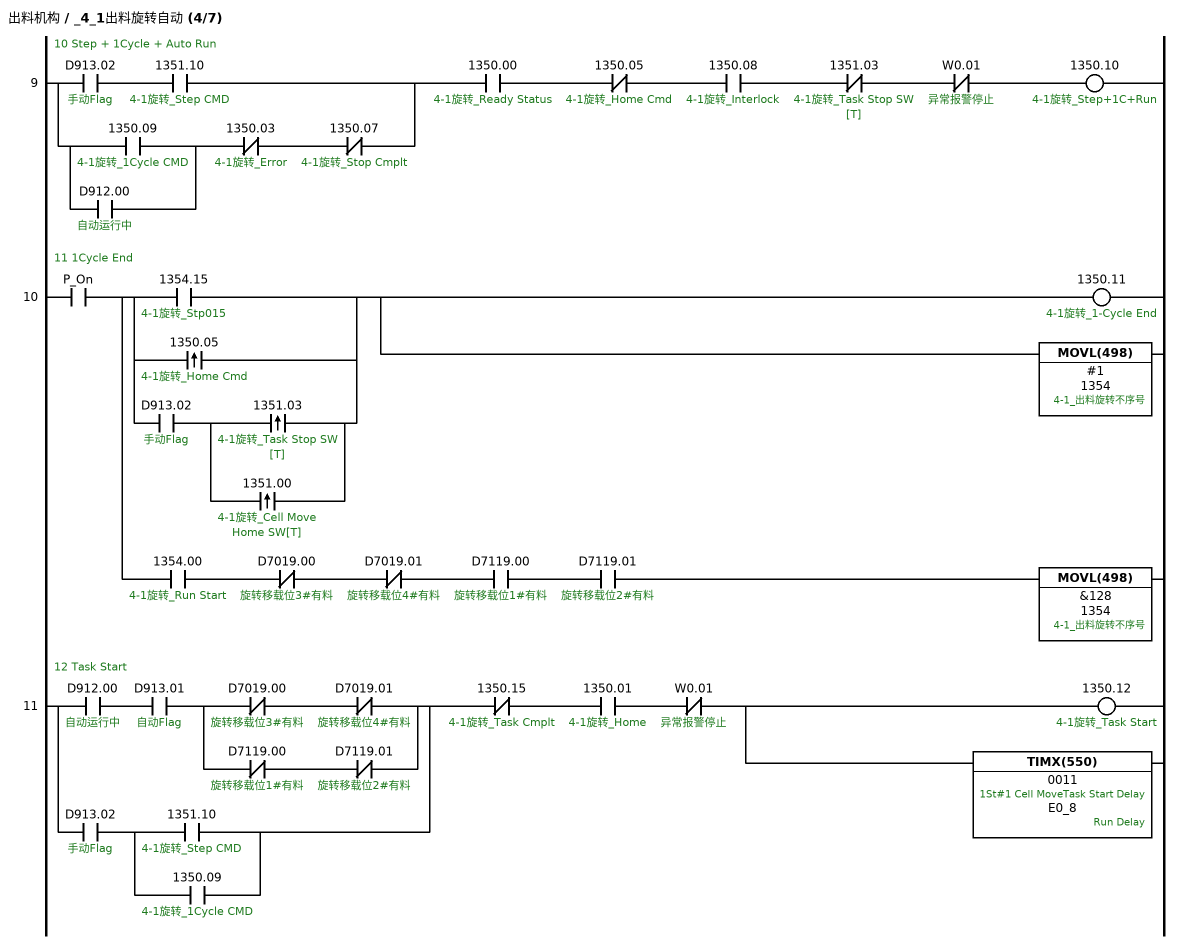
; rung 9: 10 Step + 1Cycle + Auto Run
LD D913.02  ; 手动Flag
AND 1351.10  ; 4-1旋转_Step CMD
LD 1350.09  ; 4-1旋转_1Cycle CMD
OR D912.00  ; 自动运行中
ANDNOT 1350.03  ; 4-1旋转_Error
ANDNOT 1350.07  ; 4-1旋转_Stop Cmplt
ORLD
AND 1350.00  ; 4-1旋转_Ready Status
ANDNOT 1350.05  ; 4-1旋转_Home Cmd
AND 1350.08  ; 4-1旋转_Interlock
ANDNOT 1351.03  ; 4-1旋转_Task Stop SW [T]
ANDNOT W0.01  ; 异常报警停止
OUT 1350.10  ; 4-1旋转_Step+1C+Run
; rung 10: 11 1Cycle End
LD P_On
OUT TR0
LD 1354.15  ; 4-1旋转_Stp015
@OR 1350.05  ; 4-1旋转_Home Cmd
LD D913.02  ; 手动Flag
@LD 1351.03  ; 4-1旋转_Task Stop SW [T]
@OR 1351.00  ; 4-1旋转_Cell Move Home SW[T]
ANDLD
ORLD
ANDLD
OUT 1350.11  ; 4-1旋转_1-Cycle End
MOVL(498) #1 1354  ; 4-1_出料旋转不序号
LD TR0
AND 1354.00  ; 4-1旋转_Run Start
ANDNOT D7019.00  ; 旋转移载位3#有料
ANDNOT D7019.01  ; 旋转移载位4#有料
AND D7119.00  ; 旋转移载位1#有料
AND D7119.01  ; 旋转移载位2#有料
MOVL(498) &128 1354  ; 4-1_出料旋转不序号
; rung 11: 12 Task Start
LD D912.00  ; 自动运行中
AND D913.01  ; 自动Flag
LDNOT D7019.00  ; 旋转移载位3#有料
ANDNOT D7019.01  ; 旋转移载位4#有料
LDNOT D7119.00  ; 旋转移载位1#有料
ANDNOT D7119.01  ; 旋转移载位2#有料
ORLD
ANDLD
LD D913.02  ; 手动Flag
LD 1351.10  ; 4-1旋转_Step CMD
OR 1350.09  ; 4-1旋转_1Cycle CMD
ANDLD
ORLD
ANDNOT 1350.15  ; 4-1旋转_Task Cmplt
AND 1350.01  ; 4-1旋转_Home
ANDNOT W0.01  ; 异常报警停止
OUT 1350.12  ; 4-1旋转_Task Start
TIMX(550) 0011 E0_8  ; Run Delay, 1St#1 Cell MoveTask Start Delay

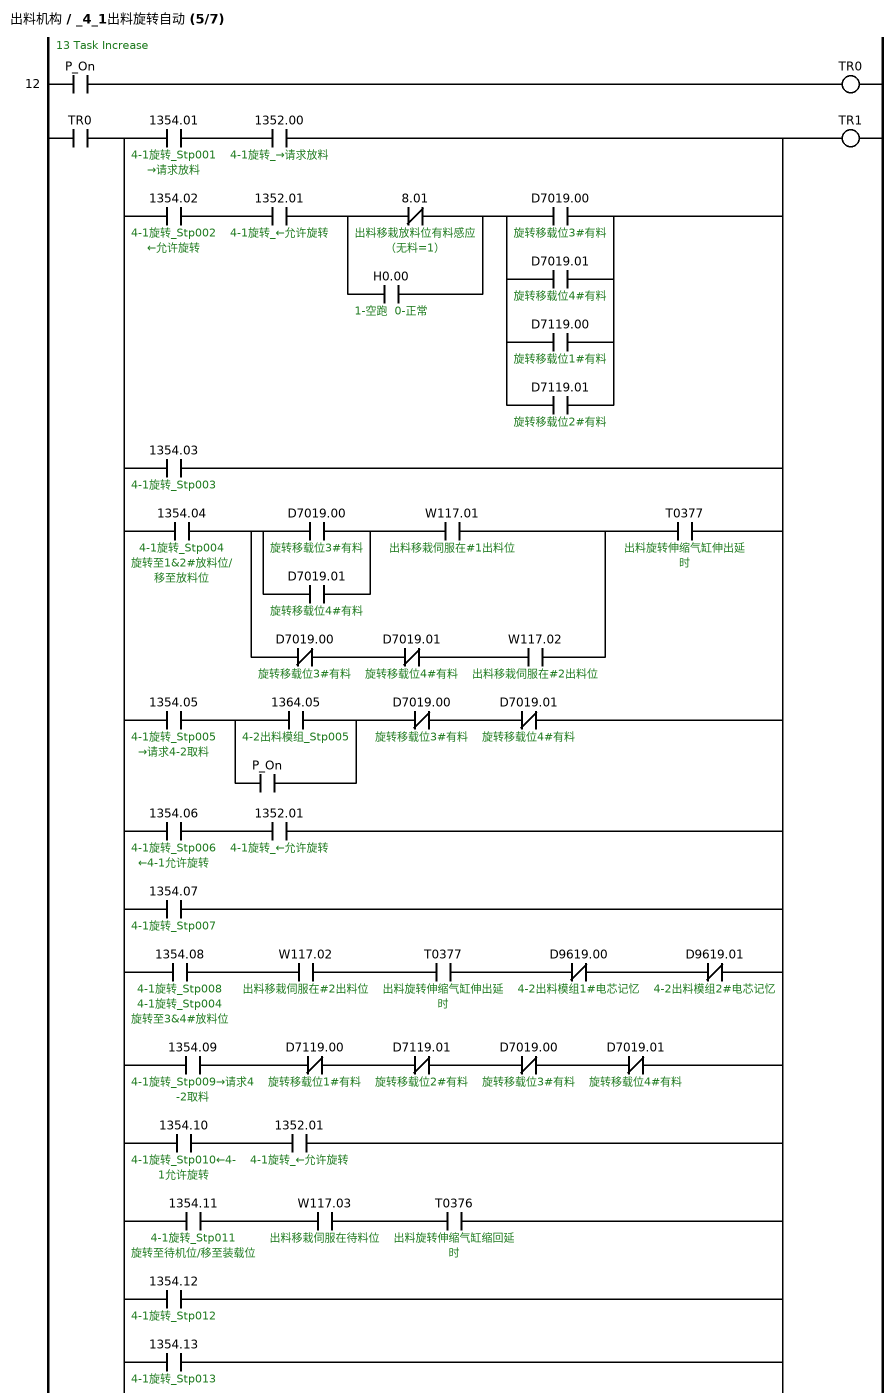

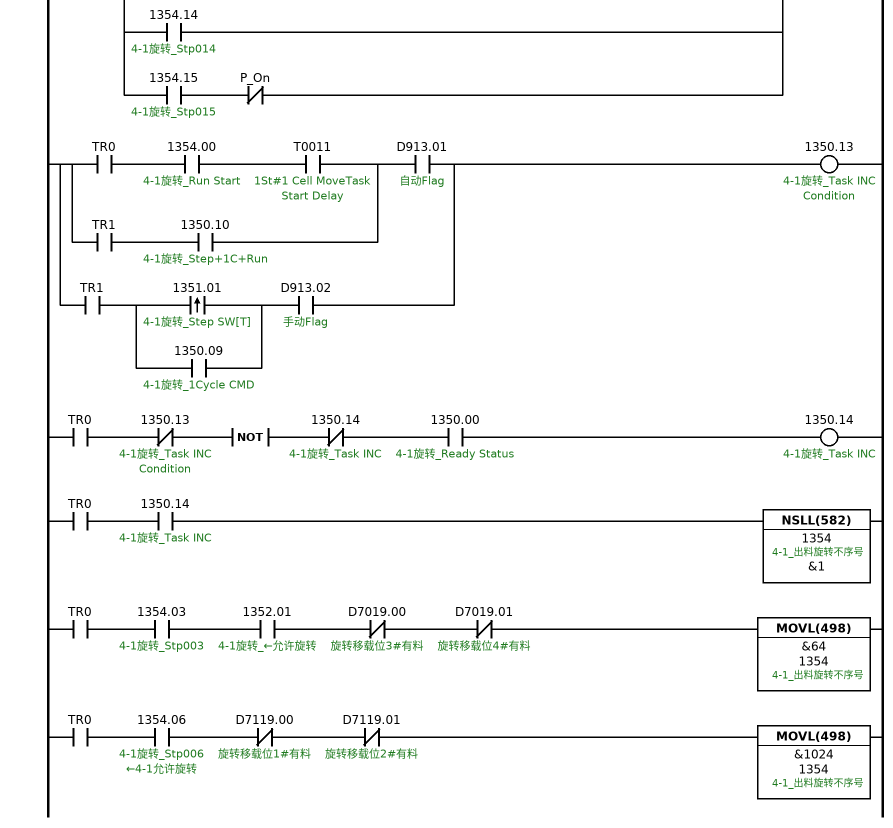
; rung 12: 13 Task Increase
LD P_On
OUT TR0
AND 1354.00  ; 4-1旋转_Run Start
AND T0011  ; 1St#1 Cell MoveTask Start Delay
LD TR0
LD 1354.01  ; 4-1旋转_Stp001 →请求放料
AND 1352.00  ; 4-1旋转_→请求放料
LD 1354.02  ; 4-1旋转_Stp002 ←允许旋转
AND 1352.01  ; 4-1旋转_←允许旋转
LDNOT 8.01  ; 出料移栽放料位有料感应（无料=1）
OR H0.00  ; 1-空跑  0-正常
ANDLD
LD D7019.00  ; 旋转移载位3#有料
OR D7019.01  ; 旋转移载位4#有料
OR D7119.00  ; 旋转移载位1#有料
OR D7119.01  ; 旋转移载位2#有料
ANDLD
ORLD
OR 1354.03  ; 4-1旋转_Stp003
LD 1354.04  ; 4-1旋转_Stp004 旋转至1&2#放料位/移至放料位
LD D7019.00  ; 旋转移载位3#有料
OR D7019.01  ; 旋转移载位4#有料
AND W117.01  ; 出料移栽伺服在#1出料位
LDNOT D7019.00  ; 旋转移载位3#有料
ANDNOT D7019.01  ; 旋转移载位4#有料
AND W117.02  ; 出料移栽伺服在#2出料位
ORLD
ANDLD
AND T0377  ; 出料旋转伸缩气缸伸出延时
ORLD
LD 1354.05  ; 4-1旋转_Stp005 →请求4-2取料
LD 1364.05  ; 4-2出料模组_Stp005  // 会停止时会出现死机现象，需确定1364.05在此处意义？
OR P_On
ANDLD
ANDNOT D7019.00  ; 旋转移载位3#有料
ANDNOT D7019.01  ; 旋转移载位4#有料
ORLD
LD 1354.06  ; 4-1旋转_Stp006 ←4-1允许旋转
AND 1352.01  ; 4-1旋转_←允许旋转
ORLD
OR 1354.07  ; 4-1旋转_Stp007
LD 1354.08  ; 4-1旋转_Stp008 4-1旋转_Stp004 旋转至3&4#放料位
AND W117.02  ; 出料移栽伺服在#2出料位
AND T0377  ; 出料旋转伸缩气缸伸出延时
ANDNOT D9619.00  ; 4-2出料模组1#电芯记忆
ANDNOT D9619.01  ; 4-2出料模组2#电芯记忆
ORLD
LD 1354.09  ; 4-1旋转_Stp009→请求4-2取料
ANDNOT D7119.00  ; 旋转移载位1#有料
ANDNOT D7119.01  ; 旋转移载位2#有料
ANDNOT D7019.00  ; 旋转移载位3#有料
ANDNOT D7019.01  ; 旋转移载位4#有料
ORLD
LD 1354.10  ; 4-1旋转_Stp010←4-1允许旋转
AND 1352.01  ; 4-1旋转_←允许旋转
ORLD
LD 1354.11  ; 4-1旋转_Stp011 旋转至待机位/移至装载位
AND W117.03  ; 出料移栽伺服在待料位
AND T0376  ; 出料旋转伸缩气缸缩回延时
ORLD
OR 1354.12  ; 4-1旋转_Stp012
OR 1354.13  ; 4-1旋转_Stp013
OR 1354.14  ; 4-1旋转_Stp014
LD 1354.15  ; 4-1旋转_Stp015
ANDNOT P_On
ORLD
ANDLD
OUT TR1
AND 1350.10  ; 4-1旋转_Step+1C+Run
ORLD
AND D913.01  ; 自动Flag
LD TR1
@LD 1351.01  ; 4-1旋转_Step SW[T]
OR 1350.09  ; 4-1旋转_1Cycle CMD
ANDLD
AND D913.02  ; 手动Flag
ORLD
OUT 1350.13  ; 4-1旋转_Task INC Condition
LD TR0
ANDNOT 1350.13  ; 4-1旋转_Task INC Condition
NOT(520)
ANDNOT 1350.14  ; 4-1旋转_Task INC
AND 1350.00  ; 4-1旋转_Ready Status
OUT 1350.14  ; 4-1旋转_Task INC
LD TR0
AND 1350.14  ; 4-1旋转_Task INC
NSLL(582) 1354 &1  ; 4-1_出料旋转不序号
LD TR0
AND 1354.03  ; 4-1旋转_Stp003
AND 1352.01  ; 4-1旋转_←允许旋转
ANDNOT D7019.00  ; 旋转移载位3#有料
ANDNOT D7019.01  ; 旋转移载位4#有料
MOVL(498) &64 1354  ; 4-1_出料旋转不序号
LD TR0
AND 1354.06  ; 4-1旋转_Stp006 ←4-1允许旋转
ANDNOT D7119.00  ; 旋转移载位1#有料
ANDNOT D7119.01  ; 旋转移载位2#有料
MOVL(498) &1024 1354  ; 4-1_出料旋转不序号

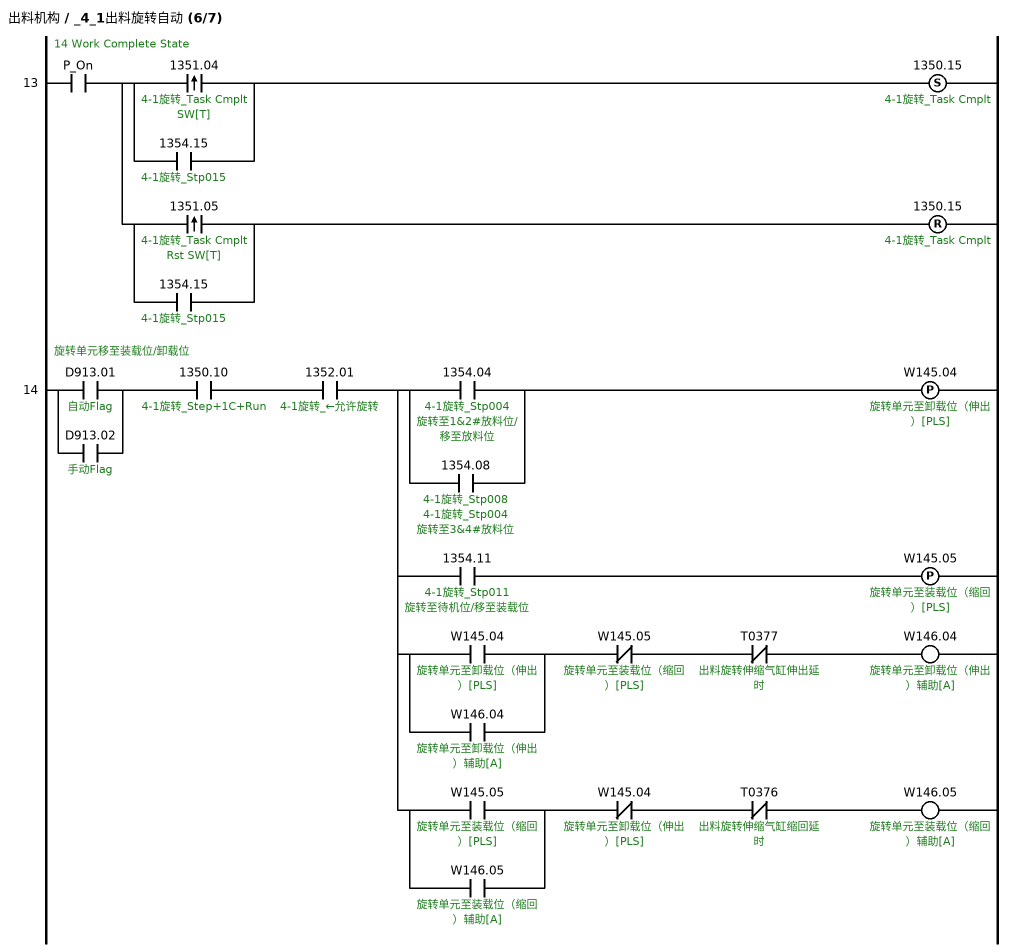
; rung 13: 14 Work Complete State
LD P_On
OUT TR0
@LD 1351.04  ; 4-1旋转_Task Cmplt SW[T]
OR 1354.15  ; 4-1旋转_Stp015
ANDLD
SET 1350.15  ; 4-1旋转_Task Cmplt
LD TR0
@LD 1351.05  ; 4-1旋转_Task Cmplt Rst SW[T]
OR 1354.15  ; 4-1旋转_Stp015
ANDLD
RSET 1350.15  ; 4-1旋转_Task Cmplt
; rung 14: 旋转单元移至装载位/卸载位
LD D913.01  ; 自动Flag
OR D913.02  ; 手动Flag
AND 1350.10  ; 4-1旋转_Step+1C+Run
AND 1352.01  ; 4-1旋转_←允许旋转
OUT TR0
LD 1354.04  ; 4-1旋转_Stp004 旋转至1&2#放料位/移至放料位
OR 1354.08  ; 4-1旋转_Stp008 4-1旋转_Stp004 旋转至3&4#放料位
ANDLD
DIFU(013) W145.04  ; 旋转单元至卸载位（伸出）[PLS]
LD TR0
AND 1354.11  ; 4-1旋转_Stp011 旋转至待机位/移至装载位
DIFU(013) W145.05  ; 旋转单元至装载位（缩回）[PLS]
LD TR0
LD W145.04  ; 旋转单元至卸载位（伸出）[PLS]
OR W146.04  ; 旋转单元至卸载位（伸出）辅助[A]
ANDLD
ANDNOT W145.05  ; 旋转单元至装载位（缩回）[PLS]
ANDNOT T0377  ; 出料旋转伸缩气缸伸出延时
OUT W146.04  ; 旋转单元至卸载位（伸出）辅助[A]
LD TR0
LD W145.05  ; 旋转单元至装载位（缩回）[PLS]
OR W146.05  ; 旋转单元至装载位（缩回）辅助[A]
ANDLD
ANDNOT W145.04  ; 旋转单元至卸载位（伸出）[PLS]
ANDNOT T0376  ; 出料旋转伸缩气缸缩回延时
OUT W146.05  ; 旋转单元至装载位（缩回）辅助[A]

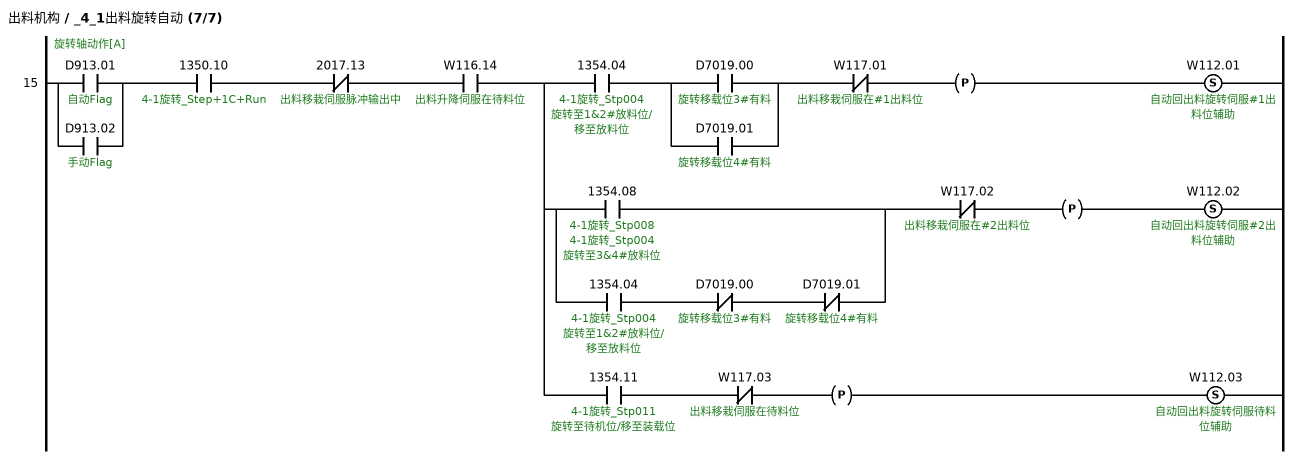
; rung 15: 旋转轴动作[A]
LD D913.01  ; 自动Flag
OR D913.02  ; 手动Flag
AND 1350.10  ; 4-1旋转_Step+1C+Run
ANDNOT 2017.13  ; 出料移栽伺服脉冲输出中
AND W116.14  ; 出料升降伺服在待料位
OUT TR0
AND 1354.04  ; 4-1旋转_Stp004 旋转至1&2#放料位/移至放料位
LD D7019.00  ; 旋转移载位3#有料
OR D7019.01  ; 旋转移载位4#有料
ANDLD
ANDNOT W117.01  ; 出料移栽伺服在#1出料位
UP(521)
SET W112.01  ; 自动回出料旋转伺服#1出料位辅助
LD TR0
LD 1354.08  ; 4-1旋转_Stp008 4-1旋转_Stp004 旋转至3&4#放料位
LD 1354.04  ; 4-1旋转_Stp004 旋转至1&2#放料位/移至放料位
ANDNOT D7019.00  ; 旋转移载位3#有料
ANDNOT D7019.01  ; 旋转移载位4#有料
ORLD
ANDLD
ANDNOT W117.02  ; 出料移栽伺服在#2出料位
UP(521)
SET W112.02  ; 自动回出料旋转伺服#2出料位辅助
LD TR0
AND 1354.11  ; 4-1旋转_Stp011 旋转至待机位/移至装载位
ANDNOT W117.03  ; 出料移栽伺服在待料位
UP(521)
SET W112.03  ; 自动回出料旋转伺服待料位辅助

### Section _4_2出料模组自动

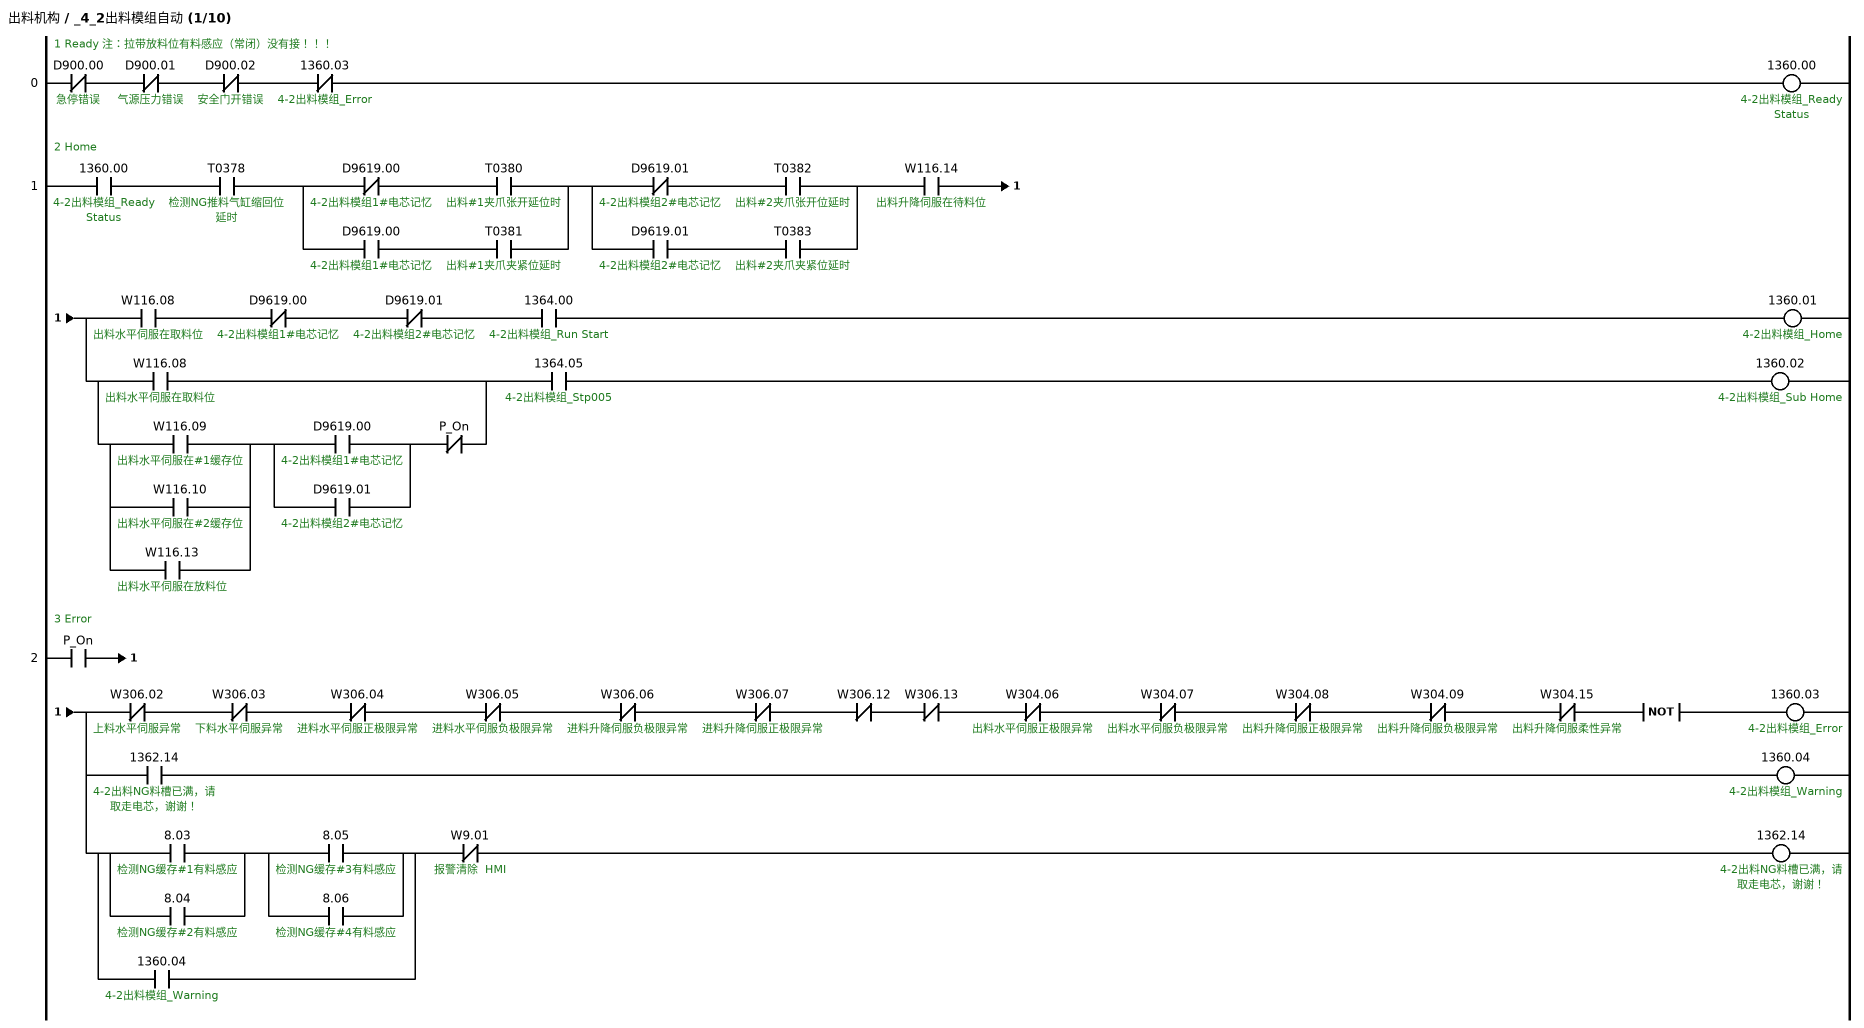
; rung 0: 1 Ready 注：拉带放料位有料感应（常闭）没有接！！！
LDNOT D900.00  ; 急停错误
ANDNOT D900.01  ; 气源压力错误
ANDNOT D900.02  ; 安全门开错误
ANDNOT 1360.03  ; 4-2出料模组_Error
OUT 1360.00  ; 4-2出料模组_Ready Status
; rung 1: 2 Home
LD 1360.00  ; 4-2出料模组_Ready Status
AND T0378  ; 检测NG推料气缸缩回位延时
LDNOT D9619.00  ; 4-2出料模组1#电芯记忆
AND T0380  ; 出料#1夹爪张开延位时
LD D9619.00  ; 4-2出料模组1#电芯记忆
AND T0381  ; 出料#1夹爪夹紧位延时
ORLD
ANDLD
LDNOT D9619.01  ; 4-2出料模组2#电芯记忆
AND T0382  ; 出料#2夹爪张开位延时
LD D9619.01  ; 4-2出料模组2#电芯记忆
AND T0383  ; 出料#2夹爪夹紧位延时
ORLD
ANDLD
AND W116.14  ; 出料升降伺服在待料位
OUT TR0
AND W116.08  ; 出料水平伺服在取料位
ANDNOT D9619.00  ; 4-2出料模组1#电芯记忆
ANDNOT D9619.01  ; 4-2出料模组2#电芯记忆
AND 1364.00  ; 4-2出料模组_Run Start
OUT 1360.01  ; 4-2出料模组_Home
LD TR0
LD W116.08  ; 出料水平伺服在取料位
LD W116.09  ; 出料水平伺服在#1缓存位
OR W116.10  ; 出料水平伺服在#2缓存位
OR W116.13  ; 出料水平伺服在放料位
LD D9619.00  ; 4-2出料模组1#电芯记忆
OR D9619.01  ; 4-2出料模组2#电芯记忆
ANDLD
ANDNOT P_On
ORLD
ANDLD
AND 1364.05  ; 4-2出料模组_Stp005
OUT 1360.02  ; 4-2出料模组_Sub Home
; rung 2: 3 Error
LD P_On
OUT TR0
ANDNOT W306.02  ; 上料水平伺服异常
ANDNOT W306.03  ; 下料水平伺服异常
ANDNOT W306.04  ; 进料水平伺服正极限异常
ANDNOT W306.05  ; 进料水平伺服负极限异常
ANDNOT W306.06  ; 进料升降伺服负极限异常
ANDNOT W306.07  ; 进料升降伺服正极限异常
ANDNOT W306.12
ANDNOT W306.13
ANDNOT W304.06  ; 出料水平伺服正极限异常
ANDNOT W304.07  ; 出料水平伺服负极限异常
ANDNOT W304.08  ; 出料升降伺服正极限异常
ANDNOT W304.09  ; 出料升降伺服负极限异常
ANDNOT W304.15  ; 出料升降伺服柔性异常
NOT(520)
OUT 1360.03  ; 4-2出料模组_Error
LD TR0
AND 1362.14  ; 4-2出料NG料槽已满，请取走电芯，谢谢！
OUT 1360.04  ; 4-2出料模组_Warning
LD TR0
LD 8.03  ; 检测NG缓存#1有料感应
OR 8.04  ; 检测NG缓存#2有料感应
LD 8.05  ; 检测NG缓存#3有料感应
OR 8.06  ; 检测NG缓存#4有料感应
ANDLD
OR 1360.04  ; 4-2出料模组_Warning
ANDLD
ANDNOT W9.01  ; 报警清除  HMI
OUT 1362.14  ; 4-2出料NG料槽已满，请取走电芯，谢谢！

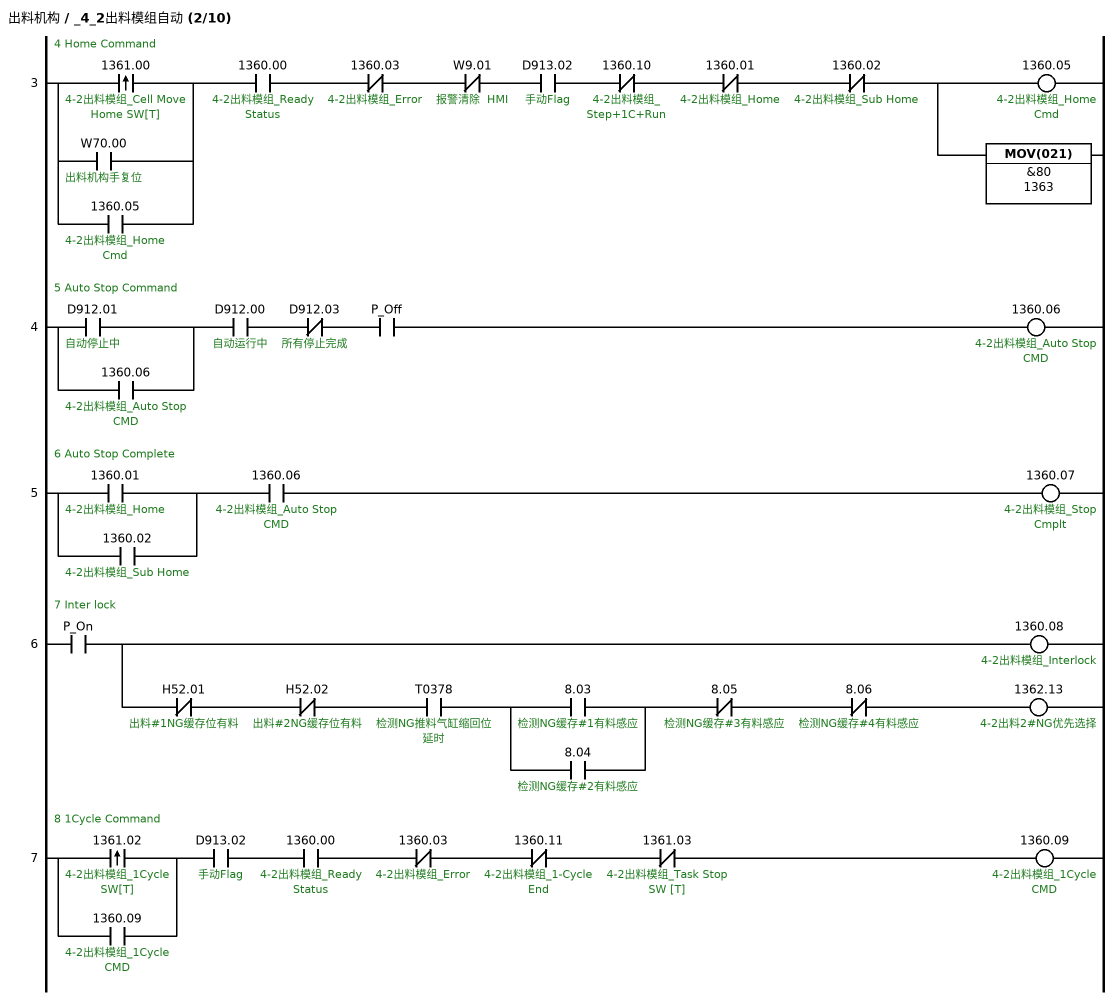
; rung 3: 4 Home Command
@LD 1361.00  ; 4-2出料模组_Cell Move Home SW[T]
OR W70.00  ; 出料机构手复位
OR 1360.05  ; 4-2出料模组_Home Cmd
AND 1360.00  ; 4-2出料模组_Ready Status
ANDNOT 1360.03  ; 4-2出料模组_Error
ANDNOT W9.01  ; 报警清除  HMI
AND D913.02  ; 手动Flag
ANDNOT 1360.10  ; 4-2出料模组_Step+1C+Run
ANDNOT 1360.01  ; 4-2出料模组_Home
ANDNOT 1360.02  ; 4-2出料模组_Sub Home
OUT 1360.05  ; 4-2出料模组_Home Cmd
MOV(021) &80 1363
; rung 4: 5 Auto Stop Command
LD D912.01  ; 自动停止中
OR 1360.06  ; 4-2出料模组_Auto Stop CMD
AND D912.00  ; 自动运行中
ANDNOT D912.03  ; 所有停止完成
AND P_Off
OUT 1360.06  ; 4-2出料模组_Auto Stop CMD
; rung 5: 6 Auto Stop Complete
LD 1360.01  ; 4-2出料模组_Home
OR 1360.02  ; 4-2出料模组_Sub Home
AND 1360.06  ; 4-2出料模组_Auto Stop CMD
OUT 1360.07  ; 4-2出料模组_Stop Cmplt
; rung 6: 7 Inter lock
LD P_On
OUT 1360.08  ; 4-2出料模组_Interlock
ANDNOT H52.01  ; 出料#1NG缓存位有料
ANDNOT H52.02  ; 出料#2NG缓存位有料
AND T0378  ; 检测NG推料气缸缩回位延时
LD 8.03  ; 检测NG缓存#1有料感应
OR 8.04  ; 检测NG缓存#2有料感应
ANDLD
ANDNOT 8.05  ; 检测NG缓存#3有料感应
ANDNOT 8.06  ; 检测NG缓存#4有料感应
OUT 1362.13  ; 4-2出料2#NG优先选择
; rung 7: 8 1Cycle Command
@LD 1361.02  ; 4-2出料模组_1Cycle SW[T]
OR 1360.09  ; 4-2出料模组_1Cycle CMD
AND D913.02  ; 手动Flag
AND 1360.00  ; 4-2出料模组_Ready Status
ANDNOT 1360.03  ; 4-2出料模组_Error
ANDNOT 1360.11  ; 4-2出料模组_1-Cycle End
ANDNOT 1361.03  ; 4-2出料模组_Task Stop SW [T]
OUT 1360.09  ; 4-2出料模组_1Cycle CMD

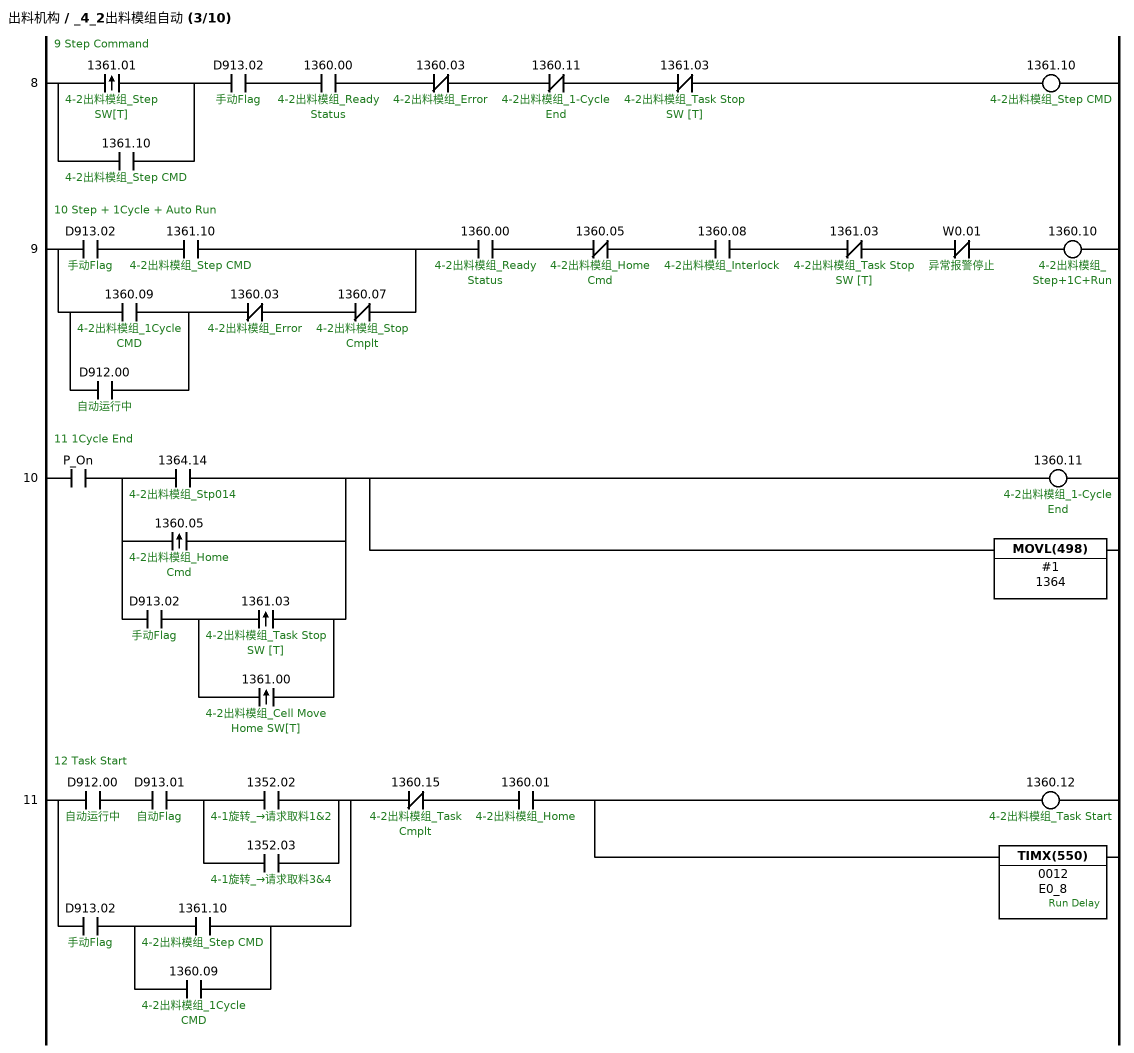
; rung 8: 9 Step Command
@LD 1361.01  ; 4-2出料模组_Step SW[T]
OR 1361.10  ; 4-2出料模组_Step CMD
AND D913.02  ; 手动Flag
AND 1360.00  ; 4-2出料模组_Ready Status
ANDNOT 1360.03  ; 4-2出料模组_Error
ANDNOT 1360.11  ; 4-2出料模组_1-Cycle End
ANDNOT 1361.03  ; 4-2出料模组_Task Stop SW [T]
OUT 1361.10  ; 4-2出料模组_Step CMD
; rung 9: 10 Step + 1Cycle + Auto Run
LD D913.02  ; 手动Flag
AND 1361.10  ; 4-2出料模组_Step CMD
LD 1360.09  ; 4-2出料模组_1Cycle CMD
OR D912.00  ; 自动运行中
ANDNOT 1360.03  ; 4-2出料模组_Error
ANDNOT 1360.07  ; 4-2出料模组_Stop Cmplt
ORLD
AND 1360.00  ; 4-2出料模组_Ready Status
ANDNOT 1360.05  ; 4-2出料模组_Home Cmd
AND 1360.08  ; 4-2出料模组_Interlock
ANDNOT 1361.03  ; 4-2出料模组_Task Stop SW [T]
ANDNOT W0.01  ; 异常报警停止
OUT 1360.10  ; 4-2出料模组_Step+1C+Run
; rung 10: 11 1Cycle End
LD P_On
LD 1364.14  ; 4-2出料模组_Stp014
@OR 1360.05  ; 4-2出料模组_Home Cmd
LD D913.02  ; 手动Flag
@LD 1361.03  ; 4-2出料模组_Task Stop SW [T]
@OR 1361.00  ; 4-2出料模组_Cell Move Home SW[T]
ANDLD
ORLD
ANDLD
OUT 1360.11  ; 4-2出料模组_1-Cycle End
MOVL(498) #1 1364
; rung 11: 12 Task Start
LD D912.00  ; 自动运行中
AND D913.01  ; 自动Flag
LD 1352.02  ; 4-1旋转_→请求取料1&2
OR 1352.03  ; 4-1旋转_→请求取料3&4
ANDLD
LD D913.02  ; 手动Flag
LD 1361.10  ; 4-2出料模组_Step CMD
OR 1360.09  ; 4-2出料模组_1Cycle CMD
ANDLD
ORLD
ANDNOT 1360.15  ; 4-2出料模组_Task Cmplt
AND 1360.01  ; 4-2出料模组_Home
OUT 1360.12  ; 4-2出料模组_Task Start
TIMX(550) 0012 E0_8  ; Run Delay

